// TIA Portal V19 export
FUNCTION_BLOCK "PositioningMachine_FB"   // FB24, LAD
TITLE = POSITIONING MACHINE
// stored: Access Published, MemoryReserve 100, SetENOAutomatically false
   VAR_INPUT
      AreaInterface : "AreaInterface";
      ZSI : "udt_ZoneSafetyInterface";
      DSI : "udt_DeviceSafetyInterface";
      Drive : "TAx_DriveInterface";
      DataIn : "PositioningMachine_DataIn";
      CIn : "PositioningMachine_CIn";
      Config : "PositioningMachine_Config";
      OL_CL_Space : LReal := 0.0;   // Limite rispetto allo spazio mancante per cambio da Move vel a Move pos abs
   END_VAR
   VAR_OUTPUT
      MachineInterface : "MachineInterface";
      DataOut : "PositioningMachine_DataOut";
      COut : "PositioningMachine_COut";
   END_VAR
   VAR_IN_OUT
      TO_Ax : TO_PositioningAxis;
      Par : "PositioningMachine_Par";
      Pers_Data : "PositioningMachine_DataPers";
      Warning : "PositioningMachine_Wng";
      Alarm : "PositioningMachine_Alr";
   END_VAR
   VAR
      InitDone : Bool := FALSE;
      Diag : Struct
         Ax : "TO_Diagnostic";
      END_STRUCT;
      HMI : Struct
         B_Preset : Bool;
         PresetPosition : LReal;
         TargetPosition : LReal;
      END_STRUCT;
      Sts : Struct
         Standstill : Bool := TRUE;
         AlarmPresence : Bool := FALSE;
         WarningPresence : Bool := FALSE;
         Man_UsePositionLimits : Bool;
         Aut_UsePositionLimits : Bool;
         Gen_Cnd : Bool;
         Bwd_Cnd : Bool := FALSE;
         Fwd_Cnd : Bool := FALSE;
         InTargetPosition : Bool;
         AxisModulo : LReal;
         MissingToTarget : LReal;
         MissingToTarget_ABS : LReal;
      END_STRUCT;
      Ctrl : Struct
         StopDueDoorOpeningRequest : Bool;
         StopInPhase : Bool;
         StopProgrammed : Bool;
         StopAborting : Bool;
         Man_HighSpeed : Bool;
         Bwd_Man : Bool;
         Fwd_Man : Bool;
         MoveToPos_Man : Bool;
         Bwd_Aut : Bool;
         Fwd_Aut : Bool;
         MoveToPos_Aut : Bool;
         Fan : Bool;
         Vel : LReal;
         Acc : LReal;
         Dec : LReal;
         Jerk : LReal;
      END_STRUCT;
      EncoderSelection { ExternalAccessible := 'False'; ExternalVisible := 'False'; ExternalWritable := 'False'} : "Axis_EncoderSelection_FB";
      WritePar { S7_SetPoint := 'True'} : "Axis_WritePar_FB";
      ReloadPosition { S7_SetPoint := 'True'} : "Axis_ReloadPosition_FB";
      LoadPosition : "Axis_ManPreset_FB";
      Ax { S7_SetPoint := 'True'} : "PositioningAxis";
      TorqueLimit { S7_SetPoint := 'True'} : MC_TORQUELIMITING;
      Fan_M : "Motor";
      TON_NoPendingCmd : TON_TIME;
      TON_Feed_DelayManChangeSpeed : TON_TIME;
      TON_InTargetPosition : TON_TIME;
      TON_MissingCndBwd { S7_SetPoint := 'True'} : TON_TIME;
      TON_MissingCndFwd { S7_SetPoint := 'True'} : TON_TIME;
      TON_Fan_DelayOff : TON_TIME;
      TON_Brake_TimeOut { S7_SetPoint := 'True'} : TON_TIME;
      AUX : Struct
         PB_Bwd : Bool;
         PB_Fwd : Bool;
         PB_MoveToPos : Bool;
         B_Preset : Bool;
      END_STRUCT;
   END_VAR
   VAR_TEMP
      PE : Struct
         PB_Bwd : Bool;
         PB_Fwd : Bool;
         PB_MoveToPos : Bool;
         B_Preset : Bool;
      END_STRUCT;
      Cnd : Bool;
      Req : Bool;
      Check : Bool;
      VelMaterialMover : LReal;
      RetVal_MeasWheelCheckRotation_Man : Int;
      RetVal_MeasWheelCheckRotation_Aut : Int;
      RetVal_MeasWheelCheckMechGearRatio : Int;
      MeasWheelVelOK : Bool;
      TorqueLimit_EngUnit : LReal;
      TorqueLimit_Percentage : LReal;
      TorqueLimit_DriveUnit : LReal;
      Bwd_CheckVel : Bool;
      Fwd_CheckVel : Bool;
      Bwd_CheckPos : Bool;
      Fwd_CheckPos : Bool;
      Real_VelTarget : LReal;
      RemainingDistanceABS : LReal;
      LimitExceeds : Bool;
      NegativeTolerance : LReal;
   END_VAR
   VAR_TEMP   // added for the SCL form of the ladder/FBD networks
      _w1 : Bool;
      _w2 : Bool;
      _w3 : Bool;
   END_VAR
BEGIN

REGION Network 1 (SCL): Init
   IF NOT #InitDone THEN

       #InitDone := TRUE;

       #Pers_Data.AxisEncoderSelection_OK := FALSE;

       #Pers_Data.AxisParameters_OK := FALSE;

       #Pers_Data.AxisReloadPostion_OK := FALSE;

   END_IF;
END_REGION

REGION Network 2 (SCL): Reset
   IF #AreaInterface.RstAlarms THEN

       #Alarm.AxisNotInOperation :=

       #Alarm.BrakeTimeOut :=

       #Warning.NotAutReady :=
       #Warning.AxisNotInOperation :=
       #Warning.MissingCnd_BWD :=
       #Warning.MissingCnd_FWD := FALSE;


   END_IF;
END_REGION

REGION Network 3: Alarm motor brake timeout
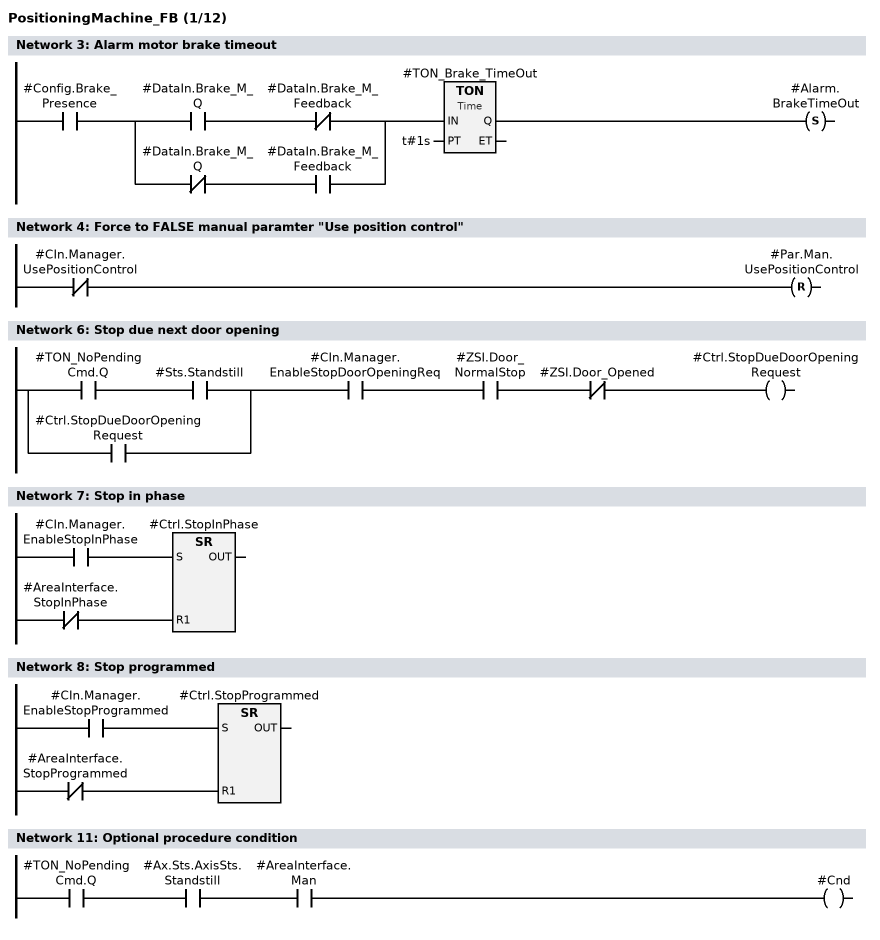
   RUNG wire#powerrail
      Contact( #Config.Brake_Presence )
      wire#w1
      Contact( #DataIn.Brake_M_Q )
      I_Contact( #DataIn.Brake_M_Feedback )
      wire#w2
      { S7_Templates := "time_type := Time" } #TON_Brake_TimeOut.TON(pt := t#1s, et =>)
      S_Coil( #Alarm.BrakeTimeOut )
   END_RUNG
   RUNG wire#w1
      I_Contact( #DataIn.Brake_M_Q )
      Contact( #DataIn.Brake_M_Feedback )
   END_RUNG wire#w2
   // the same network as SCL:
   #TON_Brake_TimeOut(IN := #Config.Brake_Presence AND ((#DataIn.Brake_M_Q AND NOT #DataIn.Brake_M_Feedback) OR (NOT #DataIn.Brake_M_Q AND #DataIn.Brake_M_Feedback)),   // TON
                      PT := t#1s);
   IF #TON_Brake_TimeOut.Q THEN #Alarm.BrakeTimeOut := TRUE; END_IF;
END_REGION

REGION Network 4: Force to FALSE manual paramter "Use position control"
   RUNG wire#powerrail
      I_Contact( #CIn.Manager.UsePositionControl )
      R_Coil( #Par.Man.UsePositionControl )
   END_RUNG
   // the same network as SCL:
   IF NOT #CIn.Manager.UsePositionControl THEN #Par.Man.UsePositionControl := FALSE; END_IF;
END_REGION

REGION Network 5: <<< MACHINE STOP >>>
END_REGION

REGION Network 6: Stop due next door opening
   RUNG wire#powerrail
      Contact( #TON_NoPendingCmd.Q )
      Contact( #Sts.Standstill )
      wire#w1
      Contact( #CIn.Manager.EnableStopDoorOpeningReq )
      Contact( #ZSI.Door_NormalStop )
      I_Contact( #ZSI.Door_Opened )
      Coil( #Ctrl.StopDueDoorOpeningRequest )
   END_RUNG
   RUNG wire#powerrail
      Contact( #Ctrl.StopDueDoorOpeningRequest )
   END_RUNG wire#w1
   // the same network as SCL:
   #Ctrl.StopDueDoorOpeningRequest := ((#TON_NoPendingCmd.Q AND #Sts.Standstill) OR #Ctrl.StopDueDoorOpeningRequest) AND #CIn.Manager.EnableStopDoorOpeningReq AND #ZSI.Door_NormalStop AND NOT #ZSI.Door_Opened;
END_REGION

REGION Network 7: Stop in phase
   RUNG wire#powerrail
      Contact( #CIn.Manager.EnableStopInPhase )
      S_SR(operand := #Ctrl.StopInPhase, r1 := wire#w1)
   END_RUNG
   RUNG wire#powerrail
      I_Contact( #AreaInterface.StopInPhase )
   END_RUNG wire#w1
   // the same network as SCL:
   IF #CIn.Manager.EnableStopInPhase THEN
       #Ctrl.StopInPhase := TRUE;   // SR flip-flop
   END_IF;
   IF NOT #AreaInterface.StopInPhase THEN #Ctrl.StopInPhase := FALSE; END_IF;
END_REGION

REGION Network 8: Stop programmed
   RUNG wire#powerrail
      Contact( #CIn.Manager.EnableStopProgrammed )
      S_SR(operand := #Ctrl.StopProgrammed, r1 := wire#w1)
   END_RUNG
   RUNG wire#powerrail
      I_Contact( #AreaInterface.StopProgrammed )
   END_RUNG wire#w1
   // the same network as SCL:
   IF #CIn.Manager.EnableStopProgrammed THEN
       #Ctrl.StopProgrammed := TRUE;   // SR flip-flop
   END_IF;
   IF NOT #AreaInterface.StopProgrammed THEN #Ctrl.StopProgrammed := FALSE; END_IF;
END_REGION

REGION Network 9: >
END_REGION

REGION Network 10: <<< OPTIONS >>>
END_REGION

REGION Network 11: Optional procedure condition
   RUNG wire#powerrail
      Contact( #TON_NoPendingCmd.Q )
      Contact( #Ax.Sts.AxisSts.Standstill )
      Contact( #AreaInterface.Man )
      Coil( #Cnd )
   END_RUNG
   // the same network as SCL:
   #Cnd := #TON_NoPendingCmd.Q AND #Ax.Sts.AxisSts.Standstill AND #AreaInterface.Man;
END_REGION

REGION Network 12: (OPTION) Motor / Measuring wheel encoder exchange
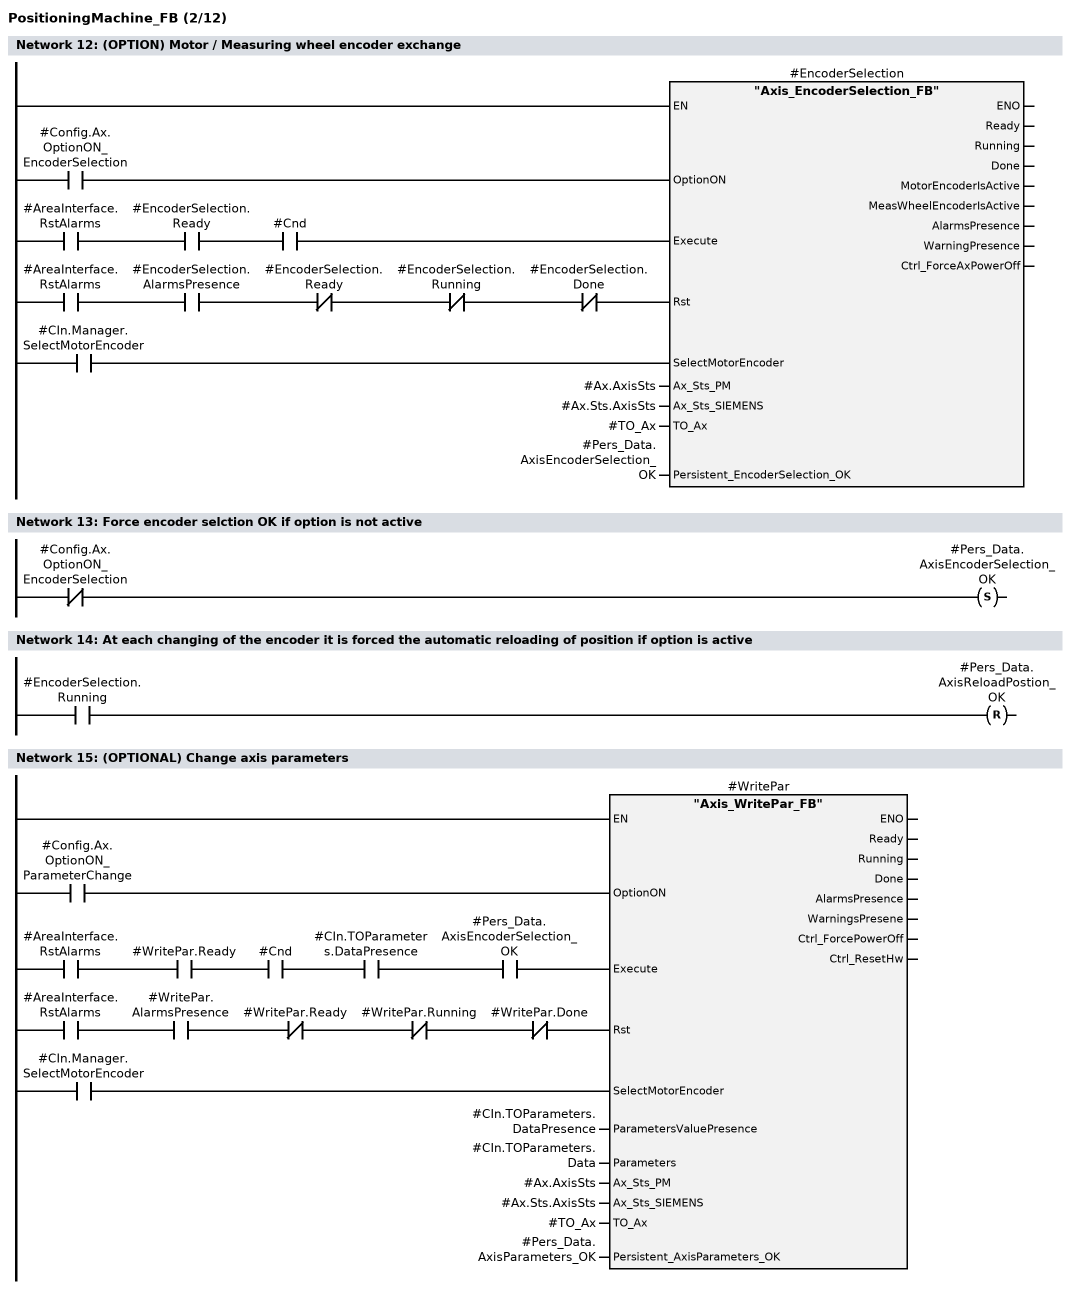
   RUNG wire#powerrail
      #EncoderSelection(OptionON := wire#w1, Execute := wire#w2, Rst := wire#w3, SelectMotorEncoder := wire#w4, Ax_Sts_PM := #Ax.AxisSts, Ax_Sts_SIEMENS := #Ax.Sts.AxisSts, TO_Ax := #TO_Ax, Persistent_EncoderSelection_OK := #Pers_Data.AxisEncoderSelection_OK, Ready =>, Running =>, Done =>, MotorEncoderIsActive =>, MeasWheelEncoderIsActive =>, AlarmsPresence =>, WarningPresence =>, Ctrl_ForceAxPowerOff =>)
   END_RUNG
   RUNG wire#powerrail
      Contact( #Config.Ax.OptionON_EncoderSelection )
   END_RUNG wire#w1
   RUNG wire#powerrail
      Contact( #AreaInterface.RstAlarms )
      Contact( #EncoderSelection.Ready )
      Contact( #Cnd )
   END_RUNG wire#w2
   RUNG wire#powerrail
      Contact( #AreaInterface.RstAlarms )
      Contact( #EncoderSelection.AlarmsPresence )
      I_Contact( #EncoderSelection.Ready )
      I_Contact( #EncoderSelection.Running )
      I_Contact( #EncoderSelection.Done )
   END_RUNG wire#w3
   RUNG wire#powerrail
      Contact( #CIn.Manager.SelectMotorEncoder )
   END_RUNG wire#w4
   // the same network as SCL:
   #EncoderSelection(OptionON := #Config.Ax.OptionON_EncoderSelection,   // "Axis_EncoderSelection_FB"
                     Execute := #AreaInterface.RstAlarms AND #EncoderSelection.Ready AND #Cnd,
                     Rst := #AreaInterface.RstAlarms AND #EncoderSelection.AlarmsPresence AND NOT #EncoderSelection.Ready AND NOT #EncoderSelection.Running AND NOT #EncoderSelection.Done,
                     SelectMotorEncoder := #CIn.Manager.SelectMotorEncoder,
                     Ax_Sts_PM := #Ax.AxisSts,
                     Ax_Sts_SIEMENS := #Ax.Sts.AxisSts,
                     TO_Ax := #TO_Ax,
                     Persistent_EncoderSelection_OK := #Pers_Data.AxisEncoderSelection_OK);
END_REGION

REGION Network 13: Force encoder selction OK if option is not active
   RUNG wire#powerrail
      I_Contact( #Config.Ax.OptionON_EncoderSelection )
      S_Coil( #Pers_Data.AxisEncoderSelection_OK )
   END_RUNG
   // the same network as SCL:
   IF NOT #Config.Ax.OptionON_EncoderSelection THEN #Pers_Data.AxisEncoderSelection_OK := TRUE; END_IF;
END_REGION

REGION Network 14: At each changing of the encoder it is forced the automatic reloading of position if option is active
   RUNG wire#powerrail
      Contact( #EncoderSelection.Running )
      R_Coil( #Pers_Data.AxisReloadPostion_OK )
   END_RUNG
   // the same network as SCL:
   IF #EncoderSelection.Running THEN #Pers_Data.AxisReloadPostion_OK := FALSE; END_IF;
END_REGION

REGION Network 15: (OPTIONAL) Change axis parameters
   RUNG wire#powerrail
      #WritePar(OptionON := wire#w1, Execute := wire#w2, Rst := wire#w3, SelectMotorEncoder := wire#w4, ParametersValuePresence := #CIn.TOParameters.DataPresence, Parameters := #CIn.TOParameters.Data, Ax_Sts_PM := #Ax.AxisSts, Ax_Sts_SIEMENS := #Ax.Sts.AxisSts, TO_Ax := #TO_Ax, Persistent_AxisParameters_OK := #Pers_Data.AxisParameters_OK, Ready =>, Running =>, Done =>, AlarmsPresence =>, WarningsPresene =>, Ctrl_ForcePowerOff =>, Ctrl_ResetHw =>)
   END_RUNG
   RUNG wire#powerrail
      Contact( #Config.Ax.OptionON_ParameterChange )
   END_RUNG wire#w1
   RUNG wire#powerrail
      Contact( #AreaInterface.RstAlarms )
      Contact( #WritePar.Ready )
      Contact( #Cnd )
      Contact( #CIn.TOParameters.DataPresence )
      Contact( #Pers_Data.AxisEncoderSelection_OK )
   END_RUNG wire#w2
   RUNG wire#powerrail
      Contact( #AreaInterface.RstAlarms )
      Contact( #WritePar.AlarmsPresence )
      I_Contact( #WritePar.Ready )
      I_Contact( #WritePar.Running )
      I_Contact( #WritePar.Done )
   END_RUNG wire#w3
   RUNG wire#powerrail
      Contact( #CIn.Manager.SelectMotorEncoder )
   END_RUNG wire#w4
   // the same network as SCL:
   #WritePar(OptionON := #Config.Ax.OptionON_ParameterChange,   // "Axis_WritePar_FB"
             Execute := #AreaInterface.RstAlarms AND #WritePar.Ready AND #Cnd AND #CIn.TOParameters.DataPresence AND #Pers_Data.AxisEncoderSelection_OK,
             Rst := #AreaInterface.RstAlarms AND #WritePar.AlarmsPresence AND NOT #WritePar.Ready AND NOT #WritePar.Running AND NOT #WritePar.Done,
             SelectMotorEncoder := #CIn.Manager.SelectMotorEncoder,
             ParametersValuePresence := #CIn.TOParameters.DataPresence,
             Parameters := #CIn.TOParameters.Data,
             Ax_Sts_PM := #Ax.AxisSts,
             Ax_Sts_SIEMENS := #Ax.Sts.AxisSts,
             TO_Ax := #TO_Ax,
             Persistent_AxisParameters_OK := #Pers_Data.AxisParameters_OK);
END_REGION

REGION Network 16: Force parameter write execution ok if option is not active
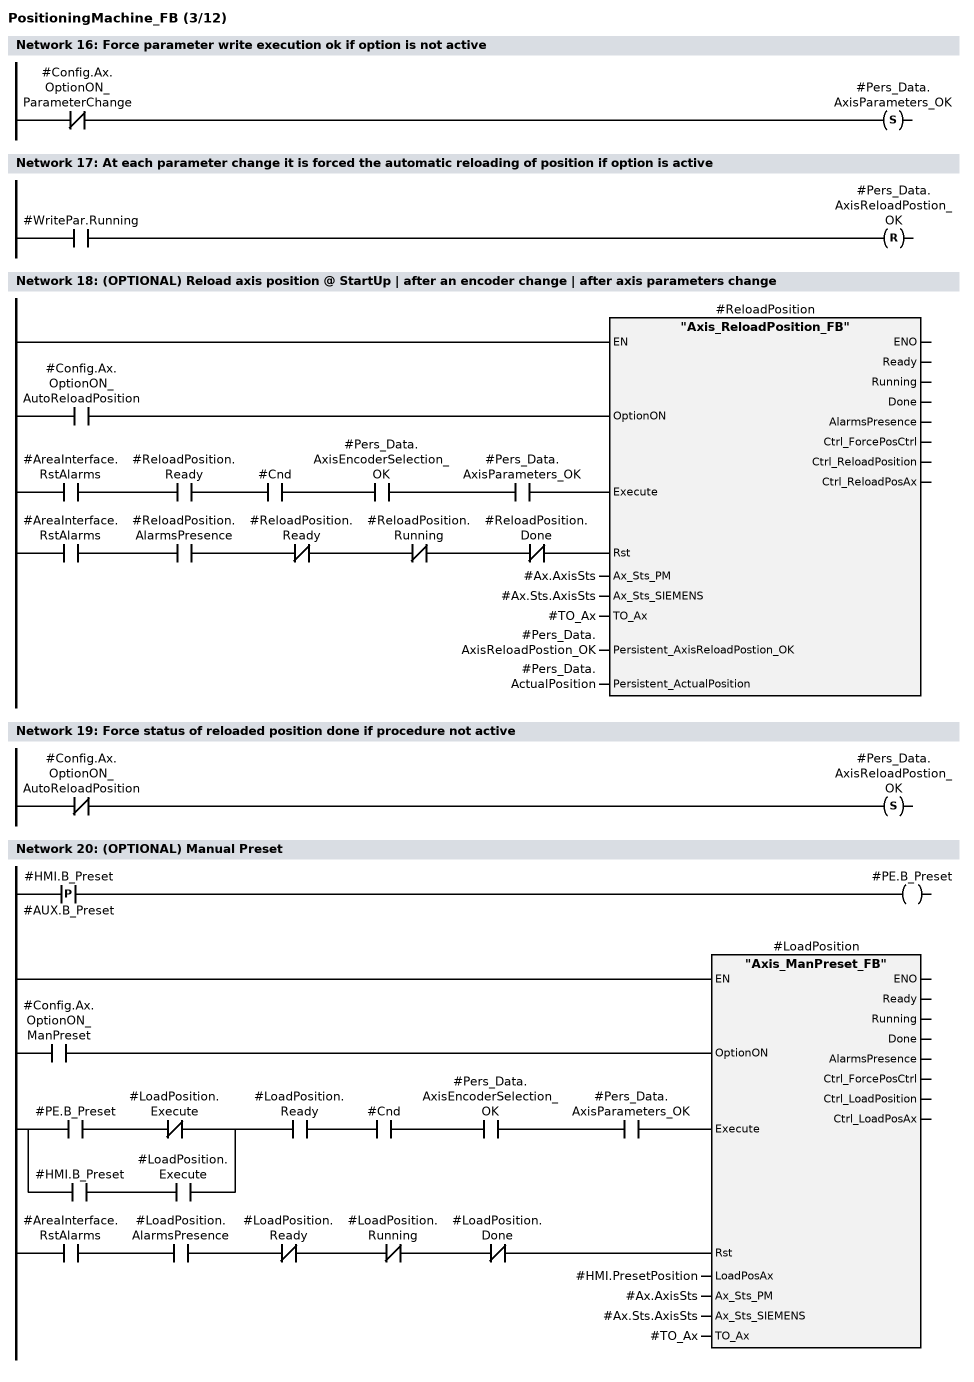
   RUNG wire#powerrail
      I_Contact( #Config.Ax.OptionON_ParameterChange )
      S_Coil( #Pers_Data.AxisParameters_OK )
   END_RUNG
   // the same network as SCL:
   IF NOT #Config.Ax.OptionON_ParameterChange THEN #Pers_Data.AxisParameters_OK := TRUE; END_IF;
END_REGION

REGION Network 17: At each parameter change it is forced the automatic reloading of position if option is active
   RUNG wire#powerrail
      Contact( #WritePar.Running )
      R_Coil( #Pers_Data.AxisReloadPostion_OK )
   END_RUNG
   // the same network as SCL:
   IF #WritePar.Running THEN #Pers_Data.AxisReloadPostion_OK := FALSE; END_IF;
END_REGION

REGION Network 18: (OPTIONAL) Reload axis position @ StartUp | after an encoder change | after axis parameters change
   RUNG wire#powerrail
      #ReloadPosition(OptionON := wire#w1, Execute := wire#w2, Rst := wire#w3, Ax_Sts_PM := #Ax.AxisSts, Ax_Sts_SIEMENS := #Ax.Sts.AxisSts, TO_Ax := #TO_Ax, Persistent_AxisReloadPostion_OK := #Pers_Data.AxisReloadPostion_OK, Persistent_ActualPosition := #Pers_Data.ActualPosition, Ready =>, Running =>, Done =>, AlarmsPresence =>, Ctrl_ForcePosCtrl =>, Ctrl_ReloadPosition =>, Ctrl_ReloadPosAx =>)
   END_RUNG
   RUNG wire#powerrail
      Contact( #Config.Ax.OptionON_AutoReloadPosition )
   END_RUNG wire#w1
   RUNG wire#powerrail
      Contact( #AreaInterface.RstAlarms )
      Contact( #ReloadPosition.Ready )
      Contact( #Cnd )
      Contact( #Pers_Data.AxisEncoderSelection_OK )
      Contact( #Pers_Data.AxisParameters_OK )
   END_RUNG wire#w2
   RUNG wire#powerrail
      Contact( #AreaInterface.RstAlarms )
      Contact( #ReloadPosition.AlarmsPresence )
      I_Contact( #ReloadPosition.Ready )
      I_Contact( #ReloadPosition.Running )
      I_Contact( #ReloadPosition.Done )
   END_RUNG wire#w3
   // the same network as SCL:
   #ReloadPosition(OptionON := #Config.Ax.OptionON_AutoReloadPosition,   // "Axis_ReloadPosition_FB"
                   Execute := #AreaInterface.RstAlarms AND #ReloadPosition.Ready AND #Cnd AND #Pers_Data.AxisEncoderSelection_OK AND #Pers_Data.AxisParameters_OK,
                   Rst := #AreaInterface.RstAlarms AND #ReloadPosition.AlarmsPresence AND NOT #ReloadPosition.Ready AND NOT #ReloadPosition.Running AND NOT #ReloadPosition.Done,
                   Ax_Sts_PM := #Ax.AxisSts,
                   Ax_Sts_SIEMENS := #Ax.Sts.AxisSts,
                   TO_Ax := #TO_Ax,
                   Persistent_AxisReloadPostion_OK := #Pers_Data.AxisReloadPostion_OK,
                   Persistent_ActualPosition := #Pers_Data.ActualPosition);
END_REGION

REGION Network 19: Force status of reloaded position done if procedure not active
   RUNG wire#powerrail
      I_Contact( #Config.Ax.OptionON_AutoReloadPosition )
      S_Coil( #Pers_Data.AxisReloadPostion_OK )
   END_RUNG
   // the same network as SCL:
   IF NOT #Config.Ax.OptionON_AutoReloadPosition THEN #Pers_Data.AxisReloadPostion_OK := TRUE; END_IF;
END_REGION

REGION Network 20: (OPTIONAL) Manual Preset
   RUNG wire#powerrail
      P_Contact(operand := #HMI.B_Preset, bit := #AUX.B_Preset)
      Coil( #PE.B_Preset )
   END_RUNG
   RUNG wire#powerrail
      #LoadPosition(OptionON := wire#w1, Execute := wire#w3, Rst := wire#w4, LoadPosAx := #HMI.PresetPosition, Ax_Sts_PM := #Ax.AxisSts, Ax_Sts_SIEMENS := #Ax.Sts.AxisSts, TO_Ax := #TO_Ax, Ready =>, Running =>, Done =>, AlarmsPresence =>, Ctrl_ForcePosCtrl =>, Ctrl_LoadPosition =>, Ctrl_LoadPosAx =>)
   END_RUNG
   RUNG wire#powerrail
      Contact( #Config.Ax.OptionON_ManPreset )
   END_RUNG wire#w1
   RUNG wire#powerrail
      Contact( #PE.B_Preset )
      I_Contact( #LoadPosition.Execute )
      wire#w2
      Contact( #LoadPosition.Ready )
      Contact( #Cnd )
      Contact( #Pers_Data.AxisEncoderSelection_OK )
      Contact( #Pers_Data.AxisParameters_OK )
   END_RUNG wire#w3
   RUNG wire#powerrail
      Contact( #HMI.B_Preset )
      Contact( #LoadPosition.Execute )
   END_RUNG wire#w2
   RUNG wire#powerrail
      Contact( #AreaInterface.RstAlarms )
      Contact( #LoadPosition.AlarmsPresence )
      I_Contact( #LoadPosition.Ready )
      I_Contact( #LoadPosition.Running )
      I_Contact( #LoadPosition.Done )
   END_RUNG wire#w4
   // the same network as SCL:
   #_w1 := #HMI.B_Preset AND NOT #AUX.B_Preset;   // rising edge of #HMI.B_Preset
   #AUX.B_Preset := #HMI.B_Preset;
   #PE.B_Preset := #_w1;
   #LoadPosition(OptionON := #Config.Ax.OptionON_ManPreset,   // "Axis_ManPreset_FB"
                 Execute := ((#PE.B_Preset AND NOT #LoadPosition.Execute) OR (#HMI.B_Preset AND #LoadPosition.Execute)) AND #LoadPosition.Ready AND #Cnd AND #Pers_Data.AxisEncoderSelection_OK AND #Pers_Data.AxisParameters_OK,
                 Rst := #AreaInterface.RstAlarms AND #LoadPosition.AlarmsPresence AND NOT #LoadPosition.Ready AND NOT #LoadPosition.Running AND NOT #LoadPosition.Done,
                 LoadPosAx := #HMI.PresetPosition,
                 Ax_Sts_PM := #Ax.AxisSts,
                 Ax_Sts_SIEMENS := #Ax.Sts.AxisSts,
                 TO_Ax := #TO_Ax);
END_REGION

REGION Network 21: At each Load position done Set Reloaad position OK
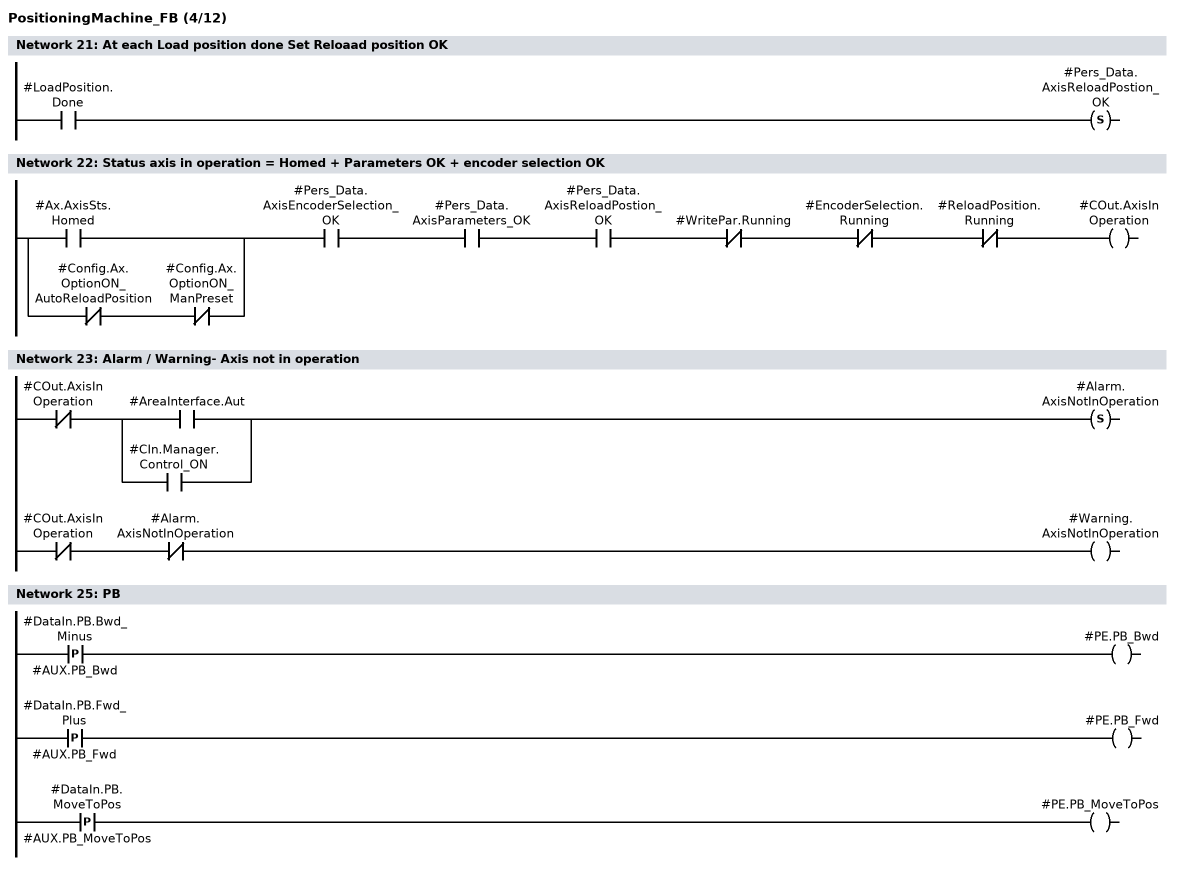
   RUNG wire#powerrail
      Contact( #LoadPosition.Done )
      S_Coil( #Pers_Data.AxisReloadPostion_OK )
   END_RUNG
   // the same network as SCL:
   IF #LoadPosition.Done THEN #Pers_Data.AxisReloadPostion_OK := TRUE; END_IF;
END_REGION

REGION Network 22: Status axis in operation = Homed + Parameters OK + encoder selection OK
   RUNG wire#powerrail
      Contact( #Ax.AxisSts.Homed )
      wire#w1
      Contact( #Pers_Data.AxisEncoderSelection_OK )
      Contact( #Pers_Data.AxisParameters_OK )
      Contact( #Pers_Data.AxisReloadPostion_OK )
      I_Contact( #WritePar.Running )
      I_Contact( #EncoderSelection.Running )
      I_Contact( #ReloadPosition.Running )
      Coil( #COut.AxisInOperation )
   END_RUNG
   RUNG wire#powerrail
      I_Contact( #Config.Ax.OptionON_AutoReloadPosition )
      I_Contact( #Config.Ax.OptionON_ManPreset )
   END_RUNG wire#w1
   // the same network as SCL:
   #COut.AxisInOperation := (#Ax.AxisSts.Homed OR (NOT #Config.Ax.OptionON_AutoReloadPosition AND NOT #Config.Ax.OptionON_ManPreset)) AND #Pers_Data.AxisEncoderSelection_OK AND #Pers_Data.AxisParameters_OK AND #Pers_Data.AxisReloadPostion_OK AND NOT #WritePar.Running AND NOT #EncoderSelection.Running AND NOT #ReloadPosition.Running;
END_REGION

REGION Network 23: Alarm / Warning- Axis not in operation
   RUNG wire#powerrail
      I_Contact( #COut.AxisInOperation )
      wire#w1
      Contact( #AreaInterface.Aut )
      wire#w2
      S_Coil( #Alarm.AxisNotInOperation )
   END_RUNG
   RUNG wire#w1
      Contact( #CIn.Manager.Control_ON )
   END_RUNG wire#w2
   RUNG wire#powerrail
      I_Contact( #COut.AxisInOperation )
      I_Contact( #Alarm.AxisNotInOperation )
      Coil( #Warning.AxisNotInOperation )
   END_RUNG
   // the same network as SCL:
   IF NOT #COut.AxisInOperation AND (#AreaInterface.Aut OR #CIn.Manager.Control_ON) THEN
       #Alarm.AxisNotInOperation := TRUE;
   END_IF;
   #Warning.AxisNotInOperation := NOT #COut.AxisInOperation AND NOT #Alarm.AxisNotInOperation;
END_REGION

REGION Network 24: <<< FEED >>>
END_REGION

REGION Network 25: PB
   RUNG wire#powerrail
      P_Contact(operand := #DataIn.PB.Bwd_Minus, bit := #AUX.PB_Bwd)
      Coil( #PE.PB_Bwd )
   END_RUNG
   RUNG wire#powerrail
      P_Contact(operand := #DataIn.PB.Fwd_Plus, bit := #AUX.PB_Fwd)
      Coil( #PE.PB_Fwd )
   END_RUNG
   RUNG wire#powerrail
      P_Contact(operand := #DataIn.PB.MoveToPos, bit := #AUX.PB_MoveToPos)
      Coil( #PE.PB_MoveToPos )
   END_RUNG
   // the same network as SCL:
   #_w1 := #DataIn.PB.Bwd_Minus AND NOT #AUX.PB_Bwd;   // rising edge of #DataIn.PB.Bwd_Minus
   #AUX.PB_Bwd := #DataIn.PB.Bwd_Minus;
   #PE.PB_Bwd := #_w1;
   #_w2 := #DataIn.PB.Fwd_Plus AND NOT #AUX.PB_Fwd;   // rising edge of #DataIn.PB.Fwd_Plus
   #AUX.PB_Fwd := #DataIn.PB.Fwd_Plus;
   #PE.PB_Fwd := #_w2;
   #_w3 := #DataIn.PB.MoveToPos AND NOT #AUX.PB_MoveToPos;   // rising edge of #DataIn.PB.MoveToPos
   #AUX.PB_MoveToPos := #DataIn.PB.MoveToPos;
   #PE.PB_MoveToPos := #_w3;
END_REGION

REGION Network 26: Man
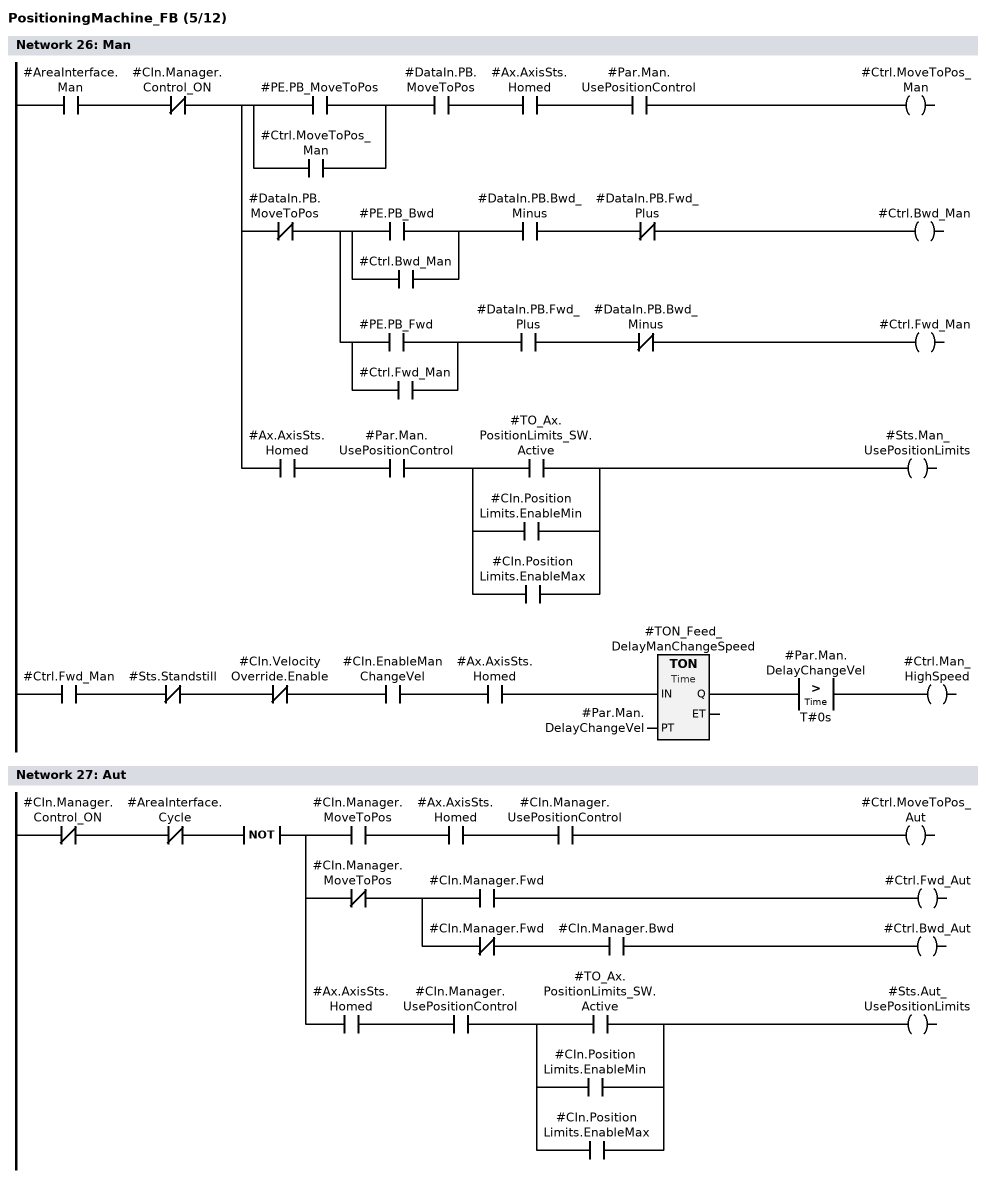
   RUNG wire#powerrail
      Contact( #AreaInterface.Man )
      I_Contact( #CIn.Manager.Control_ON )
      wire#w1
      Contact( #PE.PB_MoveToPos )
      wire#w2
      Contact( #DataIn.PB.MoveToPos )
      Contact( #Ax.AxisSts.Homed )
      Contact( #Par.Man.UsePositionControl )
      Coil( #Ctrl.MoveToPos_Man )
   END_RUNG
   RUNG wire#w1
      Contact( #Ctrl.MoveToPos_Man )
   END_RUNG wire#w2
   RUNG wire#w1
      I_Contact( #DataIn.PB.MoveToPos )
      wire#w3
      Contact( #PE.PB_Bwd )
      wire#w4
      Contact( #DataIn.PB.Bwd_Minus )
      I_Contact( #DataIn.PB.Fwd_Plus )
      Coil( #Ctrl.Bwd_Man )
   END_RUNG
   RUNG wire#w3
      Contact( #Ctrl.Bwd_Man )
   END_RUNG wire#w4
   RUNG wire#w3
      Contact( #PE.PB_Fwd )
      wire#w5
      Contact( #DataIn.PB.Fwd_Plus )
      I_Contact( #DataIn.PB.Bwd_Minus )
      Coil( #Ctrl.Fwd_Man )
   END_RUNG
   RUNG wire#w3
      Contact( #Ctrl.Fwd_Man )
   END_RUNG wire#w5
   RUNG wire#w1
      Contact( #Ax.AxisSts.Homed )
      Contact( #Par.Man.UsePositionControl )
      wire#w6
      Contact( #TO_Ax.PositionLimits_SW.Active )
      wire#w7
      Coil( #Sts.Man_UsePositionLimits )
   END_RUNG
   RUNG wire#w6
      Contact( #CIn.PositionLimits.EnableMin )
   END_RUNG wire#w7
   RUNG wire#w6
      Contact( #CIn.PositionLimits.EnableMax )
   END_RUNG wire#w7
   RUNG wire#powerrail
      Contact( #Ctrl.Fwd_Man )
      I_Contact( #Sts.Standstill )
      I_Contact( #CIn.VelocityOverride.Enable )
      Contact( #CIn.EnableManChangeVel )
      Contact( #Ax.AxisSts.Homed )
      { S7_Templates := "time_type := Time" } #TON_Feed_DelayManChangeSpeed.TON(pt := #Par.Man.DelayChangeVel, et =>)
      { S7_Templates := "SrcType := Time" } GT_Contact(in1 := #Par.Man.DelayChangeVel, in2 := T#0s)
      Coil( #Ctrl.Man_HighSpeed )
   END_RUNG
   // the same network as SCL:
   #_w1 := #AreaInterface.Man AND NOT #CIn.Manager.Control_ON;
   #Ctrl.MoveToPos_Man := #_w1 AND (#PE.PB_MoveToPos OR #Ctrl.MoveToPos_Man) AND #DataIn.PB.MoveToPos AND #Ax.AxisSts.Homed AND #Par.Man.UsePositionControl;
   #_w2 := #_w1 AND NOT #DataIn.PB.MoveToPos;
   #Ctrl.Bwd_Man := #_w2 AND (#PE.PB_Bwd OR #Ctrl.Bwd_Man) AND #DataIn.PB.Bwd_Minus AND NOT #DataIn.PB.Fwd_Plus;
   #Ctrl.Fwd_Man := #_w2 AND (#PE.PB_Fwd OR #Ctrl.Fwd_Man) AND #DataIn.PB.Fwd_Plus AND NOT #DataIn.PB.Bwd_Minus;
   #Sts.Man_UsePositionLimits := #_w1 AND #Ax.AxisSts.Homed AND #Par.Man.UsePositionControl AND (#TO_Ax.PositionLimits_SW.Active OR #CIn.PositionLimits.EnableMin OR #CIn.PositionLimits.EnableMax);
   #TON_Feed_DelayManChangeSpeed(IN := #Ctrl.Fwd_Man AND NOT #Sts.Standstill AND NOT #CIn.VelocityOverride.Enable AND #CIn.EnableManChangeVel AND #Ax.AxisSts.Homed,   // TON
                           PT := #Par.Man.DelayChangeVel);
   #Ctrl.Man_HighSpeed := #TON_Feed_DelayManChangeSpeed.Q AND (#Par.Man.DelayChangeVel > T#0s);
END_REGION

REGION Network 27: Aut
   RUNG wire#powerrail
      I_Contact( #CIn.Manager.Control_ON )
      I_Contact( #AreaInterface.Cycle )
      Not()
      wire#w1
      Contact( #CIn.Manager.MoveToPos )
      Contact( #Ax.AxisSts.Homed )
      Contact( #CIn.Manager.UsePositionControl )
      Coil( #Ctrl.MoveToPos_Aut )
   END_RUNG
   RUNG wire#w1
      I_Contact( #CIn.Manager.MoveToPos )
      wire#w2
      Contact( #CIn.Manager.Fwd )
      Coil( #Ctrl.Fwd_Aut )
   END_RUNG
   RUNG wire#w2
      I_Contact( #CIn.Manager.Fwd )
      Contact( #CIn.Manager.Bwd )
      Coil( #Ctrl.Bwd_Aut )
   END_RUNG
   RUNG wire#w1
      Contact( #Ax.AxisSts.Homed )
      Contact( #CIn.Manager.UsePositionControl )
      wire#w3
      Contact( #TO_Ax.PositionLimits_SW.Active )
      wire#w4
      Coil( #Sts.Aut_UsePositionLimits )
   END_RUNG
   RUNG wire#w3
      Contact( #CIn.PositionLimits.EnableMin )
   END_RUNG wire#w4
   RUNG wire#w3
      Contact( #CIn.PositionLimits.EnableMax )
   END_RUNG wire#w4
   // the same network as SCL:
   #_w1 := NOT (NOT #CIn.Manager.Control_ON AND NOT #AreaInterface.Cycle);
   #Ctrl.MoveToPos_Aut := #_w1 AND #CIn.Manager.MoveToPos AND #Ax.AxisSts.Homed AND #CIn.Manager.UsePositionControl;
   #_w2 := #_w1 AND NOT #CIn.Manager.MoveToPos;
   #Ctrl.Fwd_Aut := #_w2 AND #CIn.Manager.Fwd;
   #Ctrl.Bwd_Aut := #_w2 AND NOT #CIn.Manager.Fwd AND #CIn.Manager.Bwd;
   #Sts.Aut_UsePositionLimits := #_w1 AND #Ax.AxisSts.Homed AND #CIn.Manager.UsePositionControl AND (#TO_Ax.PositionLimits_SW.Active OR #CIn.PositionLimits.EnableMin OR #CIn.PositionLimits.EnableMax);
END_REGION

REGION Network 28: >
END_REGION

REGION Network 29 (SCL): Axis Modulo value; 0 If isn't a modulo axis
   #Sts.AxisModulo := 0.0;

   IF #TO_Ax.Modulo.Enable THEN
       #Sts.AxisModulo := #TO_Ax.Modulo.Length - #TO_Ax.Modulo.StartValue;
   END_IF;
END_REGION

REGION Network 30 (SCL): Position Limits
   IF #Sts.AxisModulo > 0.0 THEN

       #COut.MinPosition := #Sts.AxisModulo * 5;
       #COut.MaxPosition := #Sts.AxisModulo * 5;
   ELSE

       #COut.MinPosition := -999999999.99;
       #COut.MaxPosition := +999999999.99;

   END_IF;



   #COut.BwdMinusLsSwReached := FALSE;
   #COut.FwdPlusLsSwReached := FALSE;

   #COut.BwdMinusLimitReached := FALSE;
   #COut.FwdPlusLimitReached := FALSE;



   IF #Ax.AxisSts.Homed THEN


       //.. If software limits are enabled...
       //
       IF #TO_Ax.PositionLimits_SW.Active THEN


           // Software limit Minus reached or exceeds
           // 
           #RemainingDistanceABS := ABS("M_PosAMinusPosB"(PosA := #Pers_Data.ActualPosition, PosB := #TO_Ax.PositionLimits_SW.MinPosition, MODULE := #Sts.AxisModulo));

           #LimitExceeds := "M_CmpLT"(Xa := #Pers_Data.ActualPosition, Xb := #TO_Ax.PositionLimits_SW.MinPosition, MODULE := #Sts.AxisModulo);

           #COut.BwdMinusLsSwReached := (#RemainingDistanceABS <= #Par.PosTolerance) OR #LimitExceeds;


           // Software limit Plus reached or exceeds
           // 
           #RemainingDistanceABS := ABS("M_PosAMinusPosB"(PosA := #Pers_Data.ActualPosition, PosB := #TO_Ax.PositionLimits_SW.MaxPosition, MODULE := #Sts.AxisModulo));

           #LimitExceeds := "M_CmpGT"(Xa := #Pers_Data.ActualPosition, Xb := #TO_Ax.PositionLimits_SW.MaxPosition, MODULE := #Sts.AxisModulo);

           #COut.FwdPlusLsSwReached := (#RemainingDistanceABS <= #Par.PosTolerance) OR #LimitExceeds;



           // Set general Min / Max position limit
           // 
           #COut.MinPosition := "M_PosAPlusCostB"(PosA := #TO_Ax.PositionLimits_SW.MinPosition, CostB := (#Par.PosTolerance / 2), MODULE := #Sts.AxisModulo);
           #COut.MaxPosition := "M_PosAMinusCostB"(PosA := #TO_Ax.PositionLimits_SW.MaxPosition, CostB := (#Par.PosTolerance / 2), MODULE := #Sts.AxisModulo);

       END_IF;

       //.. IF dynamic MIN limit set..
       //
       IF #CIn.PositionLimits.EnableMin
       THEN


           #RemainingDistanceABS := ABS("M_PosAMinusPosB"(PosA := #Pers_Data.ActualPosition, PosB := #CIn.PositionLimits.PosMin, MODULE := #Sts.AxisModulo));

           #LimitExceeds := "M_CmpLT"(Xa := #Pers_Data.ActualPosition, Xb := #CIn.PositionLimits.PosMin, MODULE := #Sts.AxisModulo);

           #COut.BwdMinusLimitReached := (#RemainingDistanceABS <= #Par.PosTolerance) OR #LimitExceeds;

           // Update general MIN limit
           // 
           IF "M_CmpGT"(Xa := #CIn.PositionLimits.PosMin, Xb := #COut.MinPosition, MODULE := #Sts.AxisModulo)
           THEN
               #COut.MinPosition := #CIn.PositionLimits.PosMin;
           END_IF;
       END_IF;


       //.. IF dynamic MAX limit set..
       //
       IF #CIn.PositionLimits.EnableMax
       THEN

           #RemainingDistanceABS := ABS("M_PosAMinusPosB"(PosA := #Pers_Data.ActualPosition, PosB := #CIn.PositionLimits.PosMax, MODULE := #Sts.AxisModulo));

           #LimitExceeds := "M_CmpGT"(Xa := #Pers_Data.ActualPosition, Xb := #CIn.PositionLimits.PosMax, MODULE := #Sts.AxisModulo);

           #COut.FwdPlusLimitReached := (#RemainingDistanceABS <= #Par.PosTolerance) OR #LimitExceeds;


           // Update general MAX limit
           // 
           IF "M_CmpLT"(Xa := #CIn.PositionLimits.PosMax, Xb := #COut.MaxPosition, MODULE := #Sts.AxisModulo)
           THEN
               #COut.MaxPosition := #CIn.PositionLimits.PosMax;
           END_IF;

       END_IF;




       IF #CIn.PositionLimits.EnableMin THEN
           #COut.MinPosition := MAX(IN1 := #COut.MinPosition, IN2 := #CIn.PositionLimits.PosMin);
       END_IF;


       IF #CIn.PositionLimits.EnableMax THEN
           #COut.MaxPosition := MIN(IN1 := #COut.MaxPosition, IN2 := #CIn.PositionLimits.PosMax);
       END_IF;

   END_IF;
END_REGION

REGION Network 31 (SCL): Axis Control (Target position)
   // Move Abs parameters
   // 
   #Ax.AxisCtrl.MoveAbsDirection := 3;


   // Target position choose
   // 

   IF #CIn.Manager.Control_ON THEN

       #Ax.AxisCtrl.MoveAbsTarget := #CIn.Manager.Pos;


       IF #Ctrl.Bwd_Aut AND #Sts.Aut_UsePositionLimits THEN

           #Ax.AxisCtrl.MoveAbsTarget := #COut.MinPosition;

       ELSIF #Ctrl.Fwd_Aut AND #Sts.Aut_UsePositionLimits THEN

           #Ax.AxisCtrl.MoveAbsTarget := #COut.MinPosition;
       END_IF;

       #HMI.TargetPosition := #Ax.AxisCtrl.MoveAbsTarget;


   ELSIF #Ctrl.MoveToPos_Man  THEN

       #Ax.AxisCtrl.MoveAbsTarget := #HMI.TargetPosition;


   ELSIF #Ctrl.Bwd_Man AND #Sts.Man_UsePositionLimits THEN

       #Ax.AxisCtrl.MoveAbsTarget := #COut.MinPosition;
       #HMI.TargetPosition := #Ax.AxisCtrl.MoveAbsTarget;

   ELSIF #Ctrl.Fwd_Man AND #Sts.Man_UsePositionLimits THEN

       #Ax.AxisCtrl.MoveAbsTarget := #COut.MaxPosition;
       #HMI.TargetPosition := #Ax.AxisCtrl.MoveAbsTarget;

   END_IF;


   // Check Target position within limits
   //

   IF #Sts.Man_UsePositionLimits OR #Sts.Aut_UsePositionLimits THEN


       // Target position exceeds MIN limit
       // 
       #LimitExceeds := "M_CmpLT"(Xa := #Ax.AxisCtrl.MoveAbsTarget, Xb := #COut.MinPosition, MODULE := #Sts.AxisModulo);
       IF #LimitExceeds THEN
           #Ax.AxisCtrl.MoveAbsTarget := #COut.MinPosition;
           #HMI.TargetPosition := #Ax.AxisCtrl.MoveAbsTarget;
       END_IF;

       // Target position exceeds MAX limit
       // 
       #LimitExceeds := "M_CmpGT"(Xa := #Ax.AxisCtrl.MoveAbsTarget, Xb := #COut.MaxPosition, MODULE := #Sts.AxisModulo);
       IF #LimitExceeds THEN
           #Ax.AxisCtrl.MoveAbsTarget := #COut.MaxPosition;
           #HMI.TargetPosition := #Ax.AxisCtrl.MoveAbsTarget;
       END_IF;

   END_IF;
END_REGION

REGION Network 32 (SCL): Check missing position to reach the target
   #Sts.MissingToTarget := "M_PosAMinusPosB"(PosA := #Ax.AxisCtrl.MoveAbsTarget, PosB := #Pers_Data.ActualPosition, MODULE := #Sts.AxisModulo);

   //  Missing position to reach the target ABS value
   //  
   #Sts.MissingToTarget_ABS := ABS(#Sts.MissingToTarget);
END_REGION

REGION Network 33 (SCL): Status axis in target position

   #TON_InTargetPosition(IN := ABS(#Sts.MissingToTarget) <= #Par.PosTolerance, PT:=#Par.DelayInPosition);

   #Sts.InTargetPosition := #TON_InTargetPosition.Q AND #Ax.AxisSts.Homed AND (#Ax.AxisSts.Positioned OR NOT #Ax.AxisCtrl.MoveAbsolute);
END_REGION

REGION Network 34 (SCL): Axis Control (Velocity / Acceleration / Deceleration / Jerk)

   #COut.MaxVelocity := MIN(IN1 := #TO_Ax.DynamicLimits.MaxVelocity, IN2 := #TO_Ax.DynamicLimits.Velocity);

   #Ctrl.Vel := 0.0;


   IF #Ctrl.Bwd_Man OR #Ctrl.Fwd_Man OR #Ctrl.MoveToPos_Man THEN


       #Ctrl.Acc := #Par.Man.Acc;
       #Ctrl.Dec := #Par.Man.Dec;
       #Ctrl.Jerk := #Par.Man.Jerk;



       IF #Ctrl.Bwd_Man THEN

           #Ctrl.Vel := #Par.Man.VelBwd;

       ELSIF #Ctrl.Fwd_Man AND #Ctrl.Man_HighSpeed  THEN
           #Ctrl.Vel := #Par.Man.VelFwdHigh;

       ELSIF #Ctrl.Fwd_Man OR #Ctrl.MoveToPos_Man  THEN

           #Ctrl.Vel := #Par.Man.VelFwdLow;
       END_IF;



   ELSIF #Ctrl.MoveToPos_Aut OR #Ctrl.Bwd_Aut OR #Ctrl.Fwd_Aut  THEN

       #Ctrl.Vel := #CIn.Manager.Vel;

       #Ctrl.Acc := #CIn.Manager.Acc;
       #Ctrl.Dec := #CIn.Manager.Dec;
       #Ctrl.Jerk := #CIn.Manager.Jerk;


   END_IF;




   // Dynamic limits
   // 

   #Ctrl.Vel := MIN(IN1:=#Ctrl.Vel, IN2 := #COut.MaxVelocity);

   #Ctrl.Acc :=    MIN (IN1:=#Ctrl.Acc, IN2:= #TO_Ax.DynamicLimits.MaxAcceleration);
   IF #Ctrl.Acc <= 0.0 THEN
       #Ctrl.Acc :=  #Par.Man.Acc;
   END_IF;

   #Ctrl.Dec :=    MIN (IN1:=#Ctrl.Dec, IN2:= #TO_Ax.DynamicLimits.MaxDeceleration);
   IF #Ctrl.Dec <= 0.0 THEN
       #Ctrl.Dec :=  #Par.Man.Dec;
   END_IF;

   IF  #Ctrl.Jerk > 0.0 THEN

       #Ctrl.Jerk :=   MIN (IN1:= #Ctrl.Jerk,IN2:= #TO_Ax.DynamicLimits.MaxJerk);
   ELSE
       #Ctrl.Jerk := 0.0;
   END_IF;






   // Velocity override
   // 

   #TO_Ax.Override.Velocity := 100.0;

   IF #CIn.VelocityOverride.Enable THEN
       #TO_Ax.Override.Velocity := #CIn.VelocityOverride.Value;
   END_IF;


   // SLS velocity limit
   // 
   IF #ZSI.Door_Opened AND #Ctrl.Vel > #Config.SLS_VEL THEN
       #Ctrl.Vel := MIN(IN1:= #Ctrl.Vel, IN2:= #Config.SLS_VEL);
   END_IF;


   // Brake not open... Velocity  = 0.0
   // 
   IF #Config.Brake_Presence AND NOT #DataIn.Brake_M_Feedback THEN
       #Ctrl.Vel := 0.0;
   END_IF;

   // Init cycle force velocity = 0.0
   //
   IF #WritePar.Running OR #EncoderSelection.Running OR #ReloadPosition.Running OR #LoadPosition.Running  THEN
       #Ctrl.Vel := 0.0;
   END_IF;



   // Write dynamics value

   #Ax.AxisCtrl.Velocity :=   #Ctrl.Vel;
   #Ax.AxisCtrl.Acceleration := #Ctrl.Acc;
   #Ax.AxisCtrl.Deceleration := #Ctrl.Dec;
   #Ax.AxisCtrl.Jerk:=  #Ctrl.Jerk;
END_REGION

REGION Network 35 (SCL): Axis Control (Home Parameters) / Velocity & Dynamics
   #Ax.AxisCtrl.HomeMode := #Config.Ax.HomeMode;

   IF #ReloadPosition.Running THEN
       #Ax.AxisCtrl.HomePosition := #ReloadPosition.Ctrl_ReloadPosAx;
   ELSIF #LoadPosition.Running THEN
       #Ax.AxisCtrl.HomePosition := #LoadPosition.Ctrl_LoadPosAx;
   END_IF;
END_REGION

REGION Network 36: Move request in bwd / fwd direction case positioning
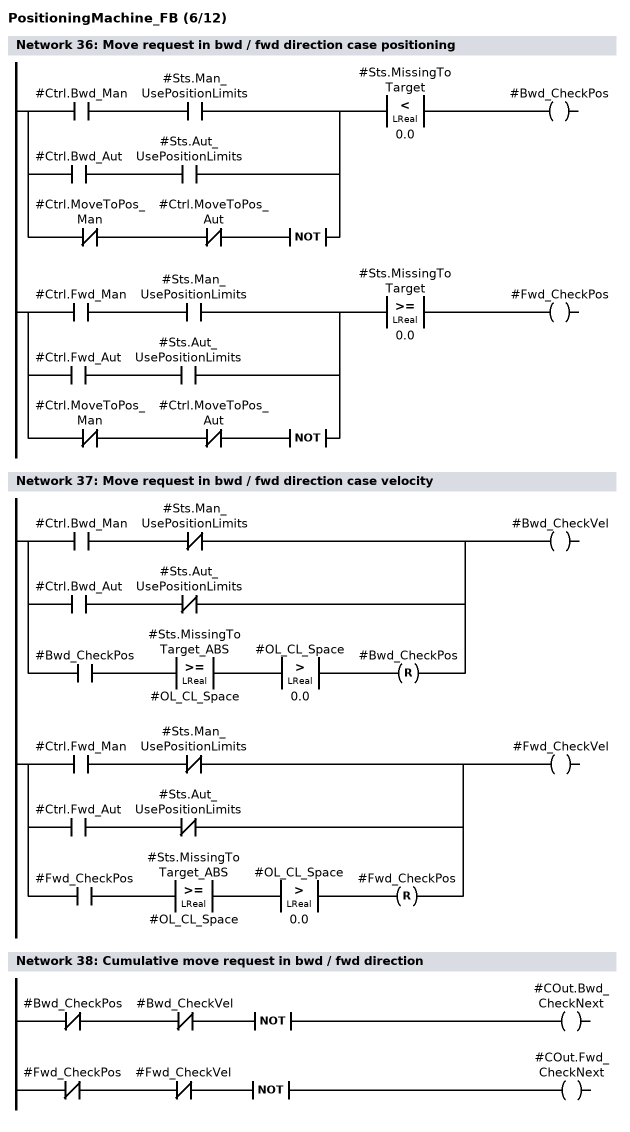
   RUNG wire#powerrail
      Contact( #Ctrl.Bwd_Man )
      Contact( #Sts.Man_UsePositionLimits )
      wire#w1
      { S7_Templates := "SrcType := LReal" } LT_Contact(in1 := #Sts.MissingToTarget, in2 := 0.0)
      Coil( #Bwd_CheckPos )
   END_RUNG
   RUNG wire#powerrail
      Contact( #Ctrl.Bwd_Aut )
      Contact( #Sts.Aut_UsePositionLimits )
   END_RUNG wire#w1
   RUNG wire#powerrail
      I_Contact( #Ctrl.MoveToPos_Man )
      I_Contact( #Ctrl.MoveToPos_Aut )
      Not()
   END_RUNG wire#w1
   RUNG wire#powerrail
      Contact( #Ctrl.Fwd_Man )
      Contact( #Sts.Man_UsePositionLimits )
      wire#w2
      { S7_Templates := "SrcType := LReal" } GE_Contact(in1 := #Sts.MissingToTarget, in2 := 0.0)
      Coil( #Fwd_CheckPos )
   END_RUNG
   RUNG wire#powerrail
      Contact( #Ctrl.Fwd_Aut )
      Contact( #Sts.Aut_UsePositionLimits )
   END_RUNG wire#w2
   RUNG wire#powerrail
      I_Contact( #Ctrl.MoveToPos_Man )
      I_Contact( #Ctrl.MoveToPos_Aut )
      Not()
   END_RUNG wire#w2
   // the same network as SCL:
   #Bwd_CheckPos := ((#Ctrl.Bwd_Man AND #Sts.Man_UsePositionLimits) OR (#Ctrl.Bwd_Aut AND #Sts.Aut_UsePositionLimits) OR NOT (NOT #Ctrl.MoveToPos_Man AND NOT #Ctrl.MoveToPos_Aut)) AND (#Sts.MissingToTarget < 0.0);
   #Fwd_CheckPos := ((#Ctrl.Fwd_Man AND #Sts.Man_UsePositionLimits) OR (#Ctrl.Fwd_Aut AND #Sts.Aut_UsePositionLimits) OR NOT (NOT #Ctrl.MoveToPos_Man AND NOT #Ctrl.MoveToPos_Aut)) AND (#Sts.MissingToTarget >= 0.0);
END_REGION

REGION Network 37: Move request in bwd / fwd direction case velocity
   RUNG wire#powerrail
      Contact( #Ctrl.Bwd_Man )
      I_Contact( #Sts.Man_UsePositionLimits )
      wire#w1
      Coil( #Bwd_CheckVel )
   END_RUNG
   RUNG wire#powerrail
      Contact( #Ctrl.Bwd_Aut )
      I_Contact( #Sts.Aut_UsePositionLimits )
   END_RUNG wire#w1
   RUNG wire#powerrail
      Contact( #Bwd_CheckPos )
      { S7_Templates := "SrcType := LReal" } GE_Contact(in1 := #Sts.MissingToTarget_ABS, in2 := #OL_CL_Space)
      { S7_Templates := "SrcType := LReal" } GT_Contact(in1 := #OL_CL_Space, in2 := 0.0)
      R_Coil( #Bwd_CheckPos )
   END_RUNG wire#w1
   RUNG wire#powerrail
      Contact( #Ctrl.Fwd_Man )
      I_Contact( #Sts.Man_UsePositionLimits )
      wire#w2
      Coil( #Fwd_CheckVel )
   END_RUNG
   RUNG wire#powerrail
      Contact( #Ctrl.Fwd_Aut )
      I_Contact( #Sts.Aut_UsePositionLimits )
   END_RUNG wire#w2
   RUNG wire#powerrail
      Contact( #Fwd_CheckPos )
      { S7_Templates := "SrcType := LReal" } GE_Contact(in1 := #Sts.MissingToTarget_ABS, in2 := #OL_CL_Space)
      { S7_Templates := "SrcType := LReal" } GT_Contact(in1 := #OL_CL_Space, in2 := 0.0)
      R_Coil( #Fwd_CheckPos )
   END_RUNG wire#w2
   // the same network as SCL:
   #_w1 := #Bwd_CheckPos AND (#Sts.MissingToTarget_ABS >= #OL_CL_Space) AND (#OL_CL_Space > 0.0);
   IF #_w1 THEN #Bwd_CheckPos := FALSE; END_IF;
   #Bwd_CheckVel := (#Ctrl.Bwd_Man AND NOT #Sts.Man_UsePositionLimits) OR (#Ctrl.Bwd_Aut AND NOT #Sts.Aut_UsePositionLimits) OR #_w1;
   #_w2 := #Fwd_CheckPos AND (#Sts.MissingToTarget_ABS >= #OL_CL_Space) AND (#OL_CL_Space > 0.0);
   IF #_w2 THEN #Fwd_CheckPos := FALSE; END_IF;
   #Fwd_CheckVel := (#Ctrl.Fwd_Man AND NOT #Sts.Man_UsePositionLimits) OR (#Ctrl.Fwd_Aut AND NOT #Sts.Aut_UsePositionLimits) OR #_w2;
END_REGION

REGION Network 38: Cumulative move request in bwd / fwd direction
   RUNG wire#powerrail
      I_Contact( #Bwd_CheckPos )
      I_Contact( #Bwd_CheckVel )
      Not()
      Coil( #COut.Bwd_CheckNext )
   END_RUNG
   RUNG wire#powerrail
      I_Contact( #Fwd_CheckPos )
      I_Contact( #Fwd_CheckVel )
      Not()
      Coil( #COut.Fwd_CheckNext )
   END_RUNG
   // the same network as SCL:
   #COut.Bwd_CheckNext := NOT (NOT #Bwd_CheckPos AND NOT #Bwd_CheckVel);
   #COut.Fwd_CheckNext := NOT (NOT #Fwd_CheckPos AND NOT #Fwd_CheckVel);
END_REGION

REGION Network 39: Conditions
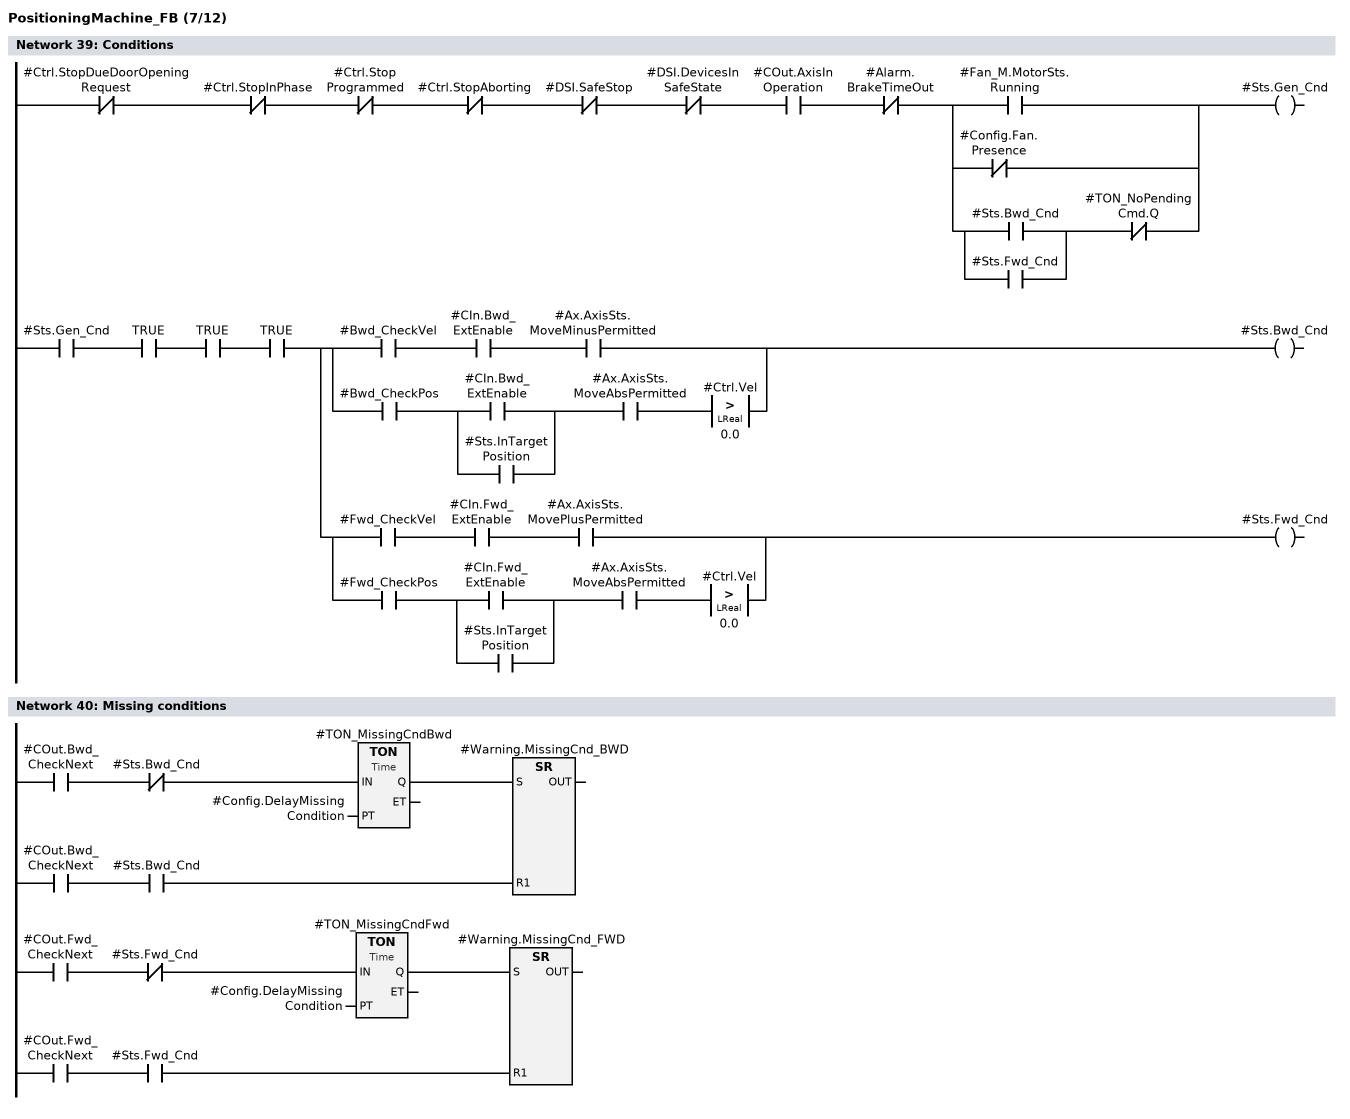
   RUNG wire#powerrail
      I_Contact( #Ctrl.StopDueDoorOpeningRequest )
      I_Contact( #Ctrl.StopInPhase )
      I_Contact( #Ctrl.StopProgrammed )
      I_Contact( #Ctrl.StopAborting )
      I_Contact( #DSI.SafeStop )
      I_Contact( #DSI.DevicesInSafeState )
      Contact( #COut.AxisInOperation )
      I_Contact( #Alarm.BrakeTimeOut )
      wire#w1
      Contact( #Fan_M.MotorSts.Running )
      wire#w2
      Coil( #Sts.Gen_Cnd )
   END_RUNG
   RUNG wire#w1
      I_Contact( #Config.Fan.Presence )
   END_RUNG wire#w2
   RUNG wire#w1
      Contact( #Sts.Bwd_Cnd )
      wire#w3
      I_Contact( #TON_NoPendingCmd.Q )
   END_RUNG wire#w2
   RUNG wire#w1
      Contact( #Sts.Fwd_Cnd )
   END_RUNG wire#w3
   RUNG wire#powerrail
      Contact( #Sts.Gen_Cnd )
      Contact( TRUE )
      Contact( TRUE )
      Contact( TRUE )
      wire#w4
      Contact( #Bwd_CheckVel )
      Contact( #CIn.Bwd_ExtEnable )
      Contact( #Ax.AxisSts.MoveMinusPermitted )
      wire#w5
      Coil( #Sts.Bwd_Cnd )
   END_RUNG
   RUNG wire#w4
      Contact( #Bwd_CheckPos )
      wire#w6
      Contact( #CIn.Bwd_ExtEnable )
      wire#w7
      Contact( #Ax.AxisSts.MoveAbsPermitted )
      { S7_Templates := "SrcType := LReal" } GT_Contact(in1 := #Ctrl.Vel, in2 := 0.0)
   END_RUNG wire#w5
   RUNG wire#w6
      Contact( #Sts.InTargetPosition )
   END_RUNG wire#w7
   RUNG wire#w4
      Contact( #Fwd_CheckVel )
      Contact( #CIn.Fwd_ExtEnable )
      Contact( #Ax.AxisSts.MovePlusPermitted )
      wire#w8
      Coil( #Sts.Fwd_Cnd )
   END_RUNG
   RUNG wire#w4
      Contact( #Fwd_CheckPos )
      wire#w9
      Contact( #CIn.Fwd_ExtEnable )
      wire#w10
      Contact( #Ax.AxisSts.MoveAbsPermitted )
      { S7_Templates := "SrcType := LReal" } GT_Contact(in1 := #Ctrl.Vel, in2 := 0.0)
   END_RUNG wire#w8
   RUNG wire#w9
      Contact( #Sts.InTargetPosition )
   END_RUNG wire#w10
   // the same network as SCL:
   #Sts.Gen_Cnd := NOT #Ctrl.StopDueDoorOpeningRequest AND NOT #Ctrl.StopInPhase AND NOT #Ctrl.StopProgrammed AND NOT #Ctrl.StopAborting AND NOT #DSI.SafeStop AND NOT #DSI.DevicesInSafeState AND #COut.AxisInOperation AND NOT #Alarm.BrakeTimeOut AND (#Fan_M.MotorSts.Running OR NOT #Config.Fan.Presence OR ((#Sts.Bwd_Cnd OR #Sts.Fwd_Cnd) AND NOT #TON_NoPendingCmd.Q));
   #_w1 := #Sts.Gen_Cnd AND TRUE AND TRUE AND TRUE;
   #Sts.Bwd_Cnd := #_w1 AND ((#Bwd_CheckVel AND #CIn.Bwd_ExtEnable AND #Ax.AxisSts.MoveMinusPermitted) OR (#Bwd_CheckPos AND (#CIn.Bwd_ExtEnable OR #Sts.InTargetPosition) AND #Ax.AxisSts.MoveAbsPermitted AND (#Ctrl.Vel > 0.0)));
   #Sts.Fwd_Cnd := #_w1 AND ((#Fwd_CheckVel AND #CIn.Fwd_ExtEnable AND #Ax.AxisSts.MovePlusPermitted) OR (#Fwd_CheckPos AND (#CIn.Fwd_ExtEnable OR #Sts.InTargetPosition) AND #Ax.AxisSts.MoveAbsPermitted AND (#Ctrl.Vel > 0.0)));
END_REGION

REGION Network 40: Missing conditions
   RUNG wire#powerrail
      Contact( #COut.Bwd_CheckNext )
      I_Contact( #Sts.Bwd_Cnd )
      { S7_Templates := "time_type := Time" } #TON_MissingCndBwd.TON(pt := #Config.DelayMissingCondition, et =>)
      S_SR(operand := #Warning.MissingCnd_BWD, r1 := wire#w1)
   END_RUNG
   RUNG wire#powerrail
      Contact( #COut.Bwd_CheckNext )
      Contact( #Sts.Bwd_Cnd )
   END_RUNG wire#w1
   RUNG wire#powerrail
      Contact( #COut.Fwd_CheckNext )
      I_Contact( #Sts.Fwd_Cnd )
      { S7_Templates := "time_type := Time" } #TON_MissingCndFwd.TON(pt := #Config.DelayMissingCondition, et =>)
      S_SR(operand := #Warning.MissingCnd_FWD, r1 := wire#w2)
   END_RUNG
   RUNG wire#powerrail
      Contact( #COut.Fwd_CheckNext )
      Contact( #Sts.Fwd_Cnd )
   END_RUNG wire#w2
   // the same network as SCL:
   #TON_MissingCndBwd(IN := #COut.Bwd_CheckNext AND NOT #Sts.Bwd_Cnd, PT := #Config.DelayMissingCondition);   // TON
   IF #TON_MissingCndBwd.Q THEN
       #Warning.MissingCnd_BWD := TRUE;   // SR flip-flop
   END_IF;
   IF #COut.Bwd_CheckNext AND #Sts.Bwd_Cnd THEN #Warning.MissingCnd_BWD := FALSE; END_IF;
   #TON_MissingCndFwd(IN := #COut.Fwd_CheckNext AND NOT #Sts.Fwd_Cnd, PT := #Config.DelayMissingCondition);   // TON
   IF #TON_MissingCndFwd.Q THEN
       #Warning.MissingCnd_FWD := TRUE;   // SR flip-flop
   END_IF;
   IF #COut.Fwd_CheckNext AND #Sts.Fwd_Cnd THEN #Warning.MissingCnd_FWD := FALSE; END_IF;
END_REGION

REGION Network 41: Axis Control (bit)
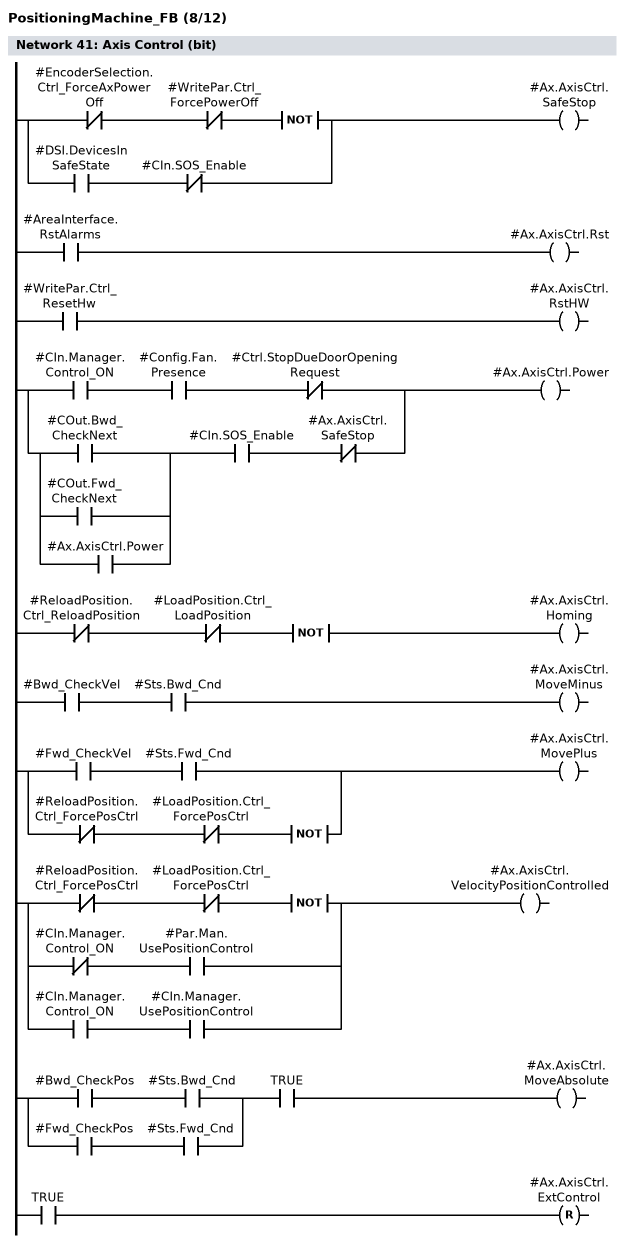
   RUNG wire#powerrail
      I_Contact( #EncoderSelection.Ctrl_ForceAxPowerOff )
      I_Contact( #WritePar.Ctrl_ForcePowerOff )
      Not()
      wire#w1
      Coil( #Ax.AxisCtrl.SafeStop )
   END_RUNG
   RUNG wire#powerrail
      Contact( #DSI.DevicesInSafeState )
      I_Contact( #CIn.SOS_Enable )
   END_RUNG wire#w1
   RUNG wire#powerrail
      Contact( #AreaInterface.RstAlarms )
      Coil( #Ax.AxisCtrl.Rst )
   END_RUNG
   RUNG wire#powerrail
      Contact( #WritePar.Ctrl_ResetHw )
      Coil( #Ax.AxisCtrl.RstHW )
   END_RUNG
   RUNG wire#powerrail
      Contact( #CIn.Manager.Control_ON )
      Contact( #Config.Fan.Presence )
      I_Contact( #Ctrl.StopDueDoorOpeningRequest )
      wire#w2
      Coil( #Ax.AxisCtrl.Power )
   END_RUNG
   RUNG wire#powerrail
      Contact( #COut.Bwd_CheckNext )
      wire#w3
      Contact( #CIn.SOS_Enable )
      I_Contact( #Ax.AxisCtrl.SafeStop )
   END_RUNG wire#w2
   RUNG wire#powerrail
      Contact( #COut.Fwd_CheckNext )
   END_RUNG wire#w3
   RUNG wire#powerrail
      Contact( #Ax.AxisCtrl.Power )
   END_RUNG wire#w3
   RUNG wire#powerrail
      I_Contact( #ReloadPosition.Ctrl_ReloadPosition )
      I_Contact( #LoadPosition.Ctrl_LoadPosition )
      Not()
      Coil( #Ax.AxisCtrl.Homing )
   END_RUNG
   RUNG wire#powerrail
      Contact( #Bwd_CheckVel )
      Contact( #Sts.Bwd_Cnd )
      Coil( #Ax.AxisCtrl.MoveMinus )
   END_RUNG
   RUNG wire#powerrail
      Contact( #Fwd_CheckVel )
      Contact( #Sts.Fwd_Cnd )
      wire#w4
      Coil( #Ax.AxisCtrl.MovePlus )
   END_RUNG
   RUNG wire#powerrail
      I_Contact( #ReloadPosition.Ctrl_ForcePosCtrl )
      I_Contact( #LoadPosition.Ctrl_ForcePosCtrl )
      Not()
   END_RUNG wire#w4
   RUNG wire#powerrail
      I_Contact( #ReloadPosition.Ctrl_ForcePosCtrl )
      I_Contact( #LoadPosition.Ctrl_ForcePosCtrl )
      Not()
      wire#w5
      Coil( #Ax.AxisCtrl.VelocityPositionControlled )
   END_RUNG
   RUNG wire#powerrail
      I_Contact( #CIn.Manager.Control_ON )
      Contact( #Par.Man.UsePositionControl )
   END_RUNG wire#w5
   RUNG wire#powerrail
      Contact( #CIn.Manager.Control_ON )
      Contact( #CIn.Manager.UsePositionControl )
   END_RUNG wire#w5
   RUNG wire#powerrail
      Contact( #Bwd_CheckPos )
      Contact( #Sts.Bwd_Cnd )
      wire#w6
      Contact( TRUE )
      Coil( #Ax.AxisCtrl.MoveAbsolute )
   END_RUNG
   RUNG wire#powerrail
      Contact( #Fwd_CheckPos )
      Contact( #Sts.Fwd_Cnd )
   END_RUNG wire#w6
   RUNG wire#powerrail
      Contact( TRUE )
      R_Coil( #Ax.AxisCtrl.ExtControl )
   END_RUNG
   // the same network as SCL:
   #Ax.AxisCtrl.SafeStop := NOT (NOT #EncoderSelection.Ctrl_ForceAxPowerOff AND NOT #WritePar.Ctrl_ForcePowerOff) OR (#DSI.DevicesInSafeState AND NOT #CIn.SOS_Enable);
   #Ax.AxisCtrl.Rst := #AreaInterface.RstAlarms;
   #Ax.AxisCtrl.RstHW := #WritePar.Ctrl_ResetHw;
   #Ax.AxisCtrl.Power := (#CIn.Manager.Control_ON AND #Config.Fan.Presence AND NOT #Ctrl.StopDueDoorOpeningRequest) OR ((#COut.Bwd_CheckNext OR #COut.Fwd_CheckNext OR #Ax.AxisCtrl.Power) AND #CIn.SOS_Enable AND NOT #Ax.AxisCtrl.SafeStop);
   #Ax.AxisCtrl.Homing := NOT (NOT #ReloadPosition.Ctrl_ReloadPosition AND NOT #LoadPosition.Ctrl_LoadPosition);
   #Ax.AxisCtrl.MoveMinus := #Bwd_CheckVel AND #Sts.Bwd_Cnd;
   #Ax.AxisCtrl.MovePlus := (#Fwd_CheckVel AND #Sts.Fwd_Cnd) OR NOT (NOT #ReloadPosition.Ctrl_ForcePosCtrl AND NOT #LoadPosition.Ctrl_ForcePosCtrl);
   #Ax.AxisCtrl.VelocityPositionControlled := NOT (NOT #ReloadPosition.Ctrl_ForcePosCtrl AND NOT #LoadPosition.Ctrl_ForcePosCtrl) OR (NOT #CIn.Manager.Control_ON AND #Par.Man.UsePositionControl) OR (#CIn.Manager.Control_ON AND #CIn.Manager.UsePositionControl);
   #Ax.AxisCtrl.MoveAbsolute := ((#Bwd_CheckPos AND #Sts.Bwd_Cnd) OR (#Fwd_CheckPos AND #Sts.Fwd_Cnd)) AND TRUE;
   IF TRUE THEN #Ax.AxisCtrl.ExtControl := FALSE; END_IF;
END_REGION

REGION Network 42: Axis manager
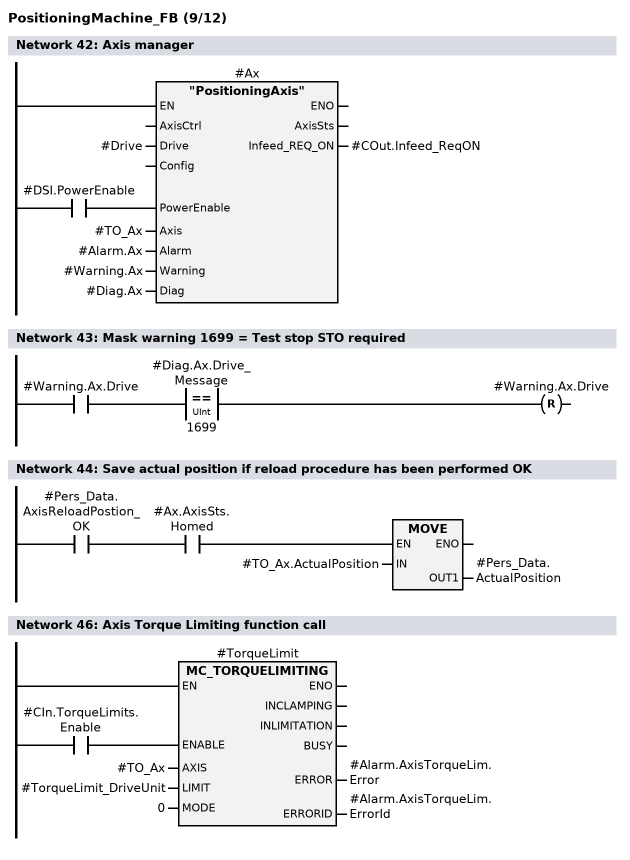
   RUNG wire#powerrail
      #Ax(PowerEnable := wire#w1, AxisCtrl :=, Drive := #Drive, Config :=, Axis := #TO_Ax, Alarm := #Alarm.Ax, Warning := #Warning.Ax, Diag := #Diag.Ax, AxisSts =>, Infeed_REQ_ON => #COut.Infeed_ReqON)
   END_RUNG
   RUNG wire#powerrail
      Contact( #DSI.PowerEnable )
   END_RUNG wire#w1
   // the same network as SCL:
   #Ax(Drive := #Drive,   // "PositioningAxis"
       PowerEnable := #DSI.PowerEnable,
       Axis := #TO_Ax,
       Alarm := #Alarm.Ax,
       Warning := #Warning.Ax,
       Diag := #Diag.Ax,
       Infeed_REQ_ON => #COut.Infeed_ReqON);
END_REGION

REGION Network 43: Mask warning 1699 = Test stop STO required
   RUNG wire#powerrail
      Contact( #Warning.Ax.Drive )
      { S7_Templates := "SrcType := UInt" } EQ_Contact(in1 := #Diag.Ax.Drive_Message, in2 := 1699)
      R_Coil( #Warning.Ax.Drive )
   END_RUNG
   // the same network as SCL:
   IF #Warning.Ax.Drive AND (#Diag.Ax.Drive_Message = 1699) THEN #Warning.Ax.Drive := FALSE; END_IF;
END_REGION

REGION Network 44: Save actual position if reload procedure has been performed OK
   RUNG wire#powerrail
      Contact( #Pers_Data.AxisReloadPostion_OK )
      Contact( #Ax.AxisSts.Homed )
      { S7_GenerateENO := "TRUE" } Move(in := #TO_Ax.ActualPosition, out1 => #Pers_Data.ActualPosition)
   END_RUNG
   // the same network as SCL:
   IF #Pers_Data.AxisReloadPostion_OK AND #Ax.AxisSts.Homed THEN
       #Pers_Data.ActualPosition := #TO_Ax.ActualPosition;
   END_IF;
END_REGION

REGION Network 45 (SCL): Axis Torque Limit normalization

   #TorqueLimit_EngUnit := LIMIT(MN:=0.0, IN:=#CIn.TorqueLimits.Value, MX:=(#TO_Ax.Actor.DriveParameter.ReferenceTorque / 2.0));

   #TorqueLimit_Percentage := #TorqueLimit_EngUnit / (#TO_Ax.Actor.DriveParameter.ReferenceTorque / 2.0)  * 100.0;

   #TorqueLimit_DriveUnit := 30720 / 100.0 * #TorqueLimit_Percentage;



   #TorqueLimit_DriveUnit := #TorqueLimit_Percentage;
END_REGION

REGION Network 46: Axis Torque Limiting function call
   RUNG wire#powerrail
      #TorqueLimit.MC_TORQUELIMITING(Enable := wire#w1, Axis := #TO_Ax, Limit := #TorqueLimit_DriveUnit, Mode := 0, InClamping =>, InLimitation =>, Busy =>, Error => #Alarm.AxisTorqueLim.Error, ErrorId => #Alarm.AxisTorqueLim.ErrorId)
   END_RUNG
   RUNG wire#powerrail
      Contact( #CIn.TorqueLimits.Enable )
   END_RUNG wire#w1
   // the same network as SCL:
   #TorqueLimit(Enable := #CIn.TorqueLimits.Enable,   // MC_TORQUELIMITING
                Axis := #TO_Ax,
                Limit := #TorqueLimit_DriveUnit,
                Mode := 0,
                Error => #Alarm.AxisTorqueLim.Error,
                ErrorId => #Alarm.AxisTorqueLim.ErrorId);
END_REGION

REGION Network 47: Coordination Out
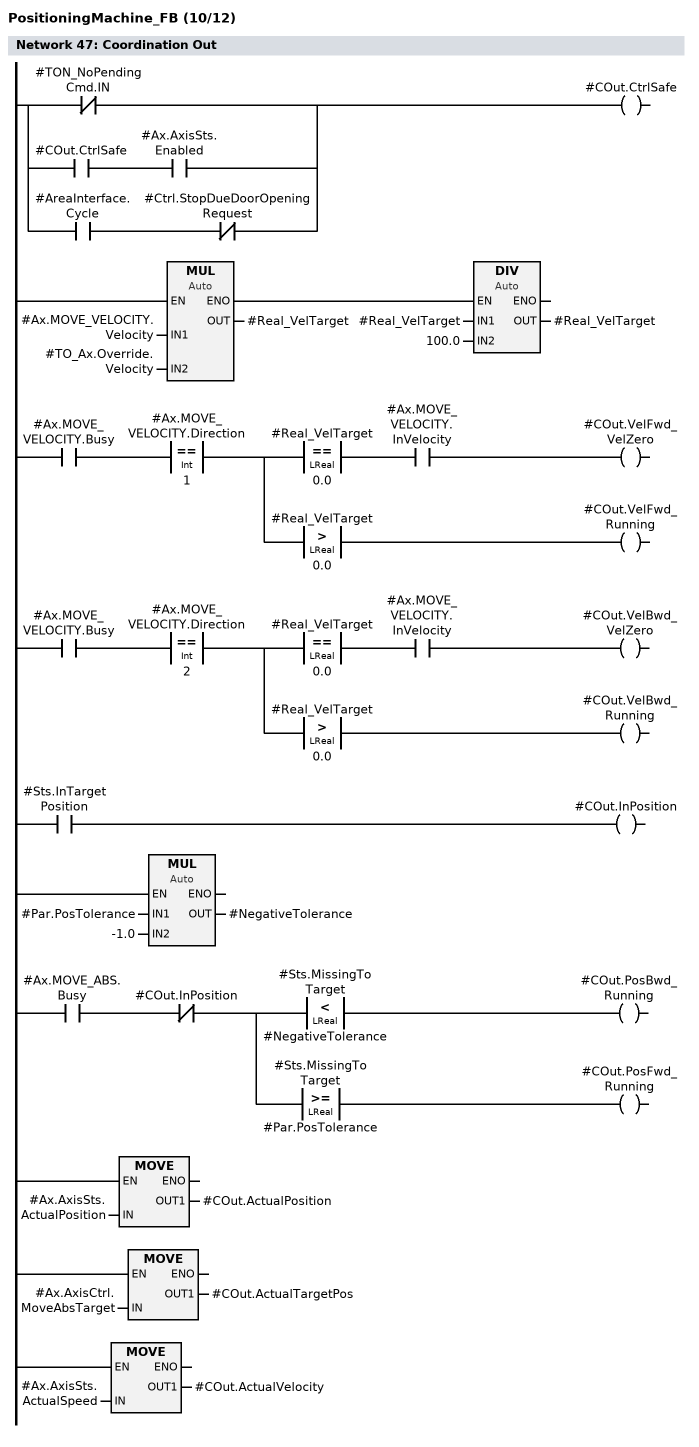
   RUNG wire#powerrail
      I_Contact( #TON_NoPendingCmd.IN )
      wire#w1
      Coil( #COut.CtrlSafe )
   END_RUNG
   RUNG wire#powerrail
      Contact( #COut.CtrlSafe )
      Contact( #Ax.AxisSts.Enabled )
   END_RUNG wire#w1
   RUNG wire#powerrail
      Contact( #AreaInterface.Cycle )
      I_Contact( #Ctrl.StopDueDoorOpeningRequest )
   END_RUNG wire#w1
   RUNG wire#powerrail
      { S7_GenerateENO := "TRUE" } Mul(in1 := #Ax.MOVE_VELOCITY.Velocity, in2 := #TO_Ax.Override.Velocity, out => #Real_VelTarget)
      { S7_GenerateENO := "TRUE" } Div(in1 := #Real_VelTarget, in2 := 100.0, out => #Real_VelTarget)
   END_RUNG
   RUNG wire#powerrail
      Contact( #Ax.MOVE_VELOCITY.Busy )
      { S7_Templates := "SrcType := Int" } EQ_Contact(in1 := #Ax.MOVE_VELOCITY.Direction, in2 := 1)
      wire#w2
      { S7_Templates := "SrcType := LReal" } EQ_Contact(in1 := #Real_VelTarget, in2 := 0.0)
      Contact( #Ax.MOVE_VELOCITY.InVelocity )
      Coil( #COut.VelFwd_VelZero )
   END_RUNG
   RUNG wire#w2
      { S7_Templates := "SrcType := LReal" } GT_Contact(in1 := #Real_VelTarget, in2 := 0.0)
      Coil( #COut.VelFwd_Running )
   END_RUNG
   RUNG wire#powerrail
      Contact( #Ax.MOVE_VELOCITY.Busy )
      { S7_Templates := "SrcType := Int" } EQ_Contact(in1 := #Ax.MOVE_VELOCITY.Direction, in2 := 2)
      wire#w3
      { S7_Templates := "SrcType := LReal" } EQ_Contact(in1 := #Real_VelTarget, in2 := 0.0)
      Contact( #Ax.MOVE_VELOCITY.InVelocity )
      Coil( #COut.VelBwd_VelZero )
   END_RUNG
   RUNG wire#w3
      { S7_Templates := "SrcType := LReal" } GT_Contact(in1 := #Real_VelTarget, in2 := 0.0)
      Coil( #COut.VelBwd_Running )
   END_RUNG
   RUNG wire#powerrail
      Contact( #Sts.InTargetPosition )
      Coil( #COut.InPosition )
   END_RUNG
   RUNG wire#powerrail
      Mul(in1 := #Par.PosTolerance, in2 := -1.0, out => #NegativeTolerance)
   END_RUNG
   RUNG wire#powerrail
      Contact( #Ax.MOVE_ABS.Busy )
      I_Contact( #COut.InPosition )
      wire#w4
      { S7_Templates := "SrcType := LReal" } LT_Contact(in1 := #Sts.MissingToTarget, in2 := #NegativeTolerance)
      Coil( #COut.PosBwd_Running )
   END_RUNG
   RUNG wire#w4
      { S7_Templates := "SrcType := LReal" } GE_Contact(in1 := #Sts.MissingToTarget, in2 := #Par.PosTolerance)
      Coil( #COut.PosFwd_Running )
   END_RUNG
   RUNG wire#powerrail
      Move(in := #Ax.AxisSts.ActualPosition, out1 => #COut.ActualPosition)
   END_RUNG
   RUNG wire#powerrail
      Move(in := #Ax.AxisCtrl.MoveAbsTarget, out1 => #COut.ActualTargetPos)
   END_RUNG
   RUNG wire#powerrail
      Move(in := #Ax.AxisSts.ActualSpeed, out1 => #COut.ActualVelocity)
   END_RUNG
   // the same network as SCL:
   // ENO of a box is taken as its EN; it also drops when the box reports an error
   #COut.CtrlSafe := NOT #TON_NoPendingCmd.IN OR (#COut.CtrlSafe AND #Ax.AxisSts.Enabled) OR (#AreaInterface.Cycle AND NOT #Ctrl.StopDueDoorOpeningRequest);
   #Real_VelTarget := #Ax.MOVE_VELOCITY.Velocity * #TO_Ax.Override.Velocity;
   #Real_VelTarget := #Real_VelTarget / 100.0;
   #_w1 := #Ax.MOVE_VELOCITY.Busy AND (#Ax.MOVE_VELOCITY.Direction = 1);
   #COut.VelFwd_VelZero := #_w1 AND (#Real_VelTarget = 0.0) AND #Ax.MOVE_VELOCITY.InVelocity;
   #COut.VelFwd_Running := #_w1 AND (#Real_VelTarget > 0.0);
   #_w2 := #Ax.MOVE_VELOCITY.Busy AND (#Ax.MOVE_VELOCITY.Direction = 2);
   #COut.VelBwd_VelZero := #_w2 AND (#Real_VelTarget = 0.0) AND #Ax.MOVE_VELOCITY.InVelocity;
   #COut.VelBwd_Running := #_w2 AND (#Real_VelTarget > 0.0);
   #COut.InPosition := #Sts.InTargetPosition;
   #NegativeTolerance := #Par.PosTolerance * (-1.0);
   #_w3 := #Ax.MOVE_ABS.Busy AND NOT #COut.InPosition;
   #COut.PosBwd_Running := #_w3 AND (#Sts.MissingToTarget < #NegativeTolerance);
   #COut.PosFwd_Running := #_w3 AND (#Sts.MissingToTarget >= #Par.PosTolerance);
   #COut.ActualPosition := #Ax.AxisSts.ActualPosition;
   #COut.ActualTargetPos := #Ax.AxisCtrl.MoveAbsTarget;
   #COut.ActualVelocity := #Ax.AxisSts.ActualSpeed;
END_REGION

REGION Network 48: >
END_REGION

REGION Network 49: <<< MOTOR FAN >>>
END_REGION

REGION Network 50: Run
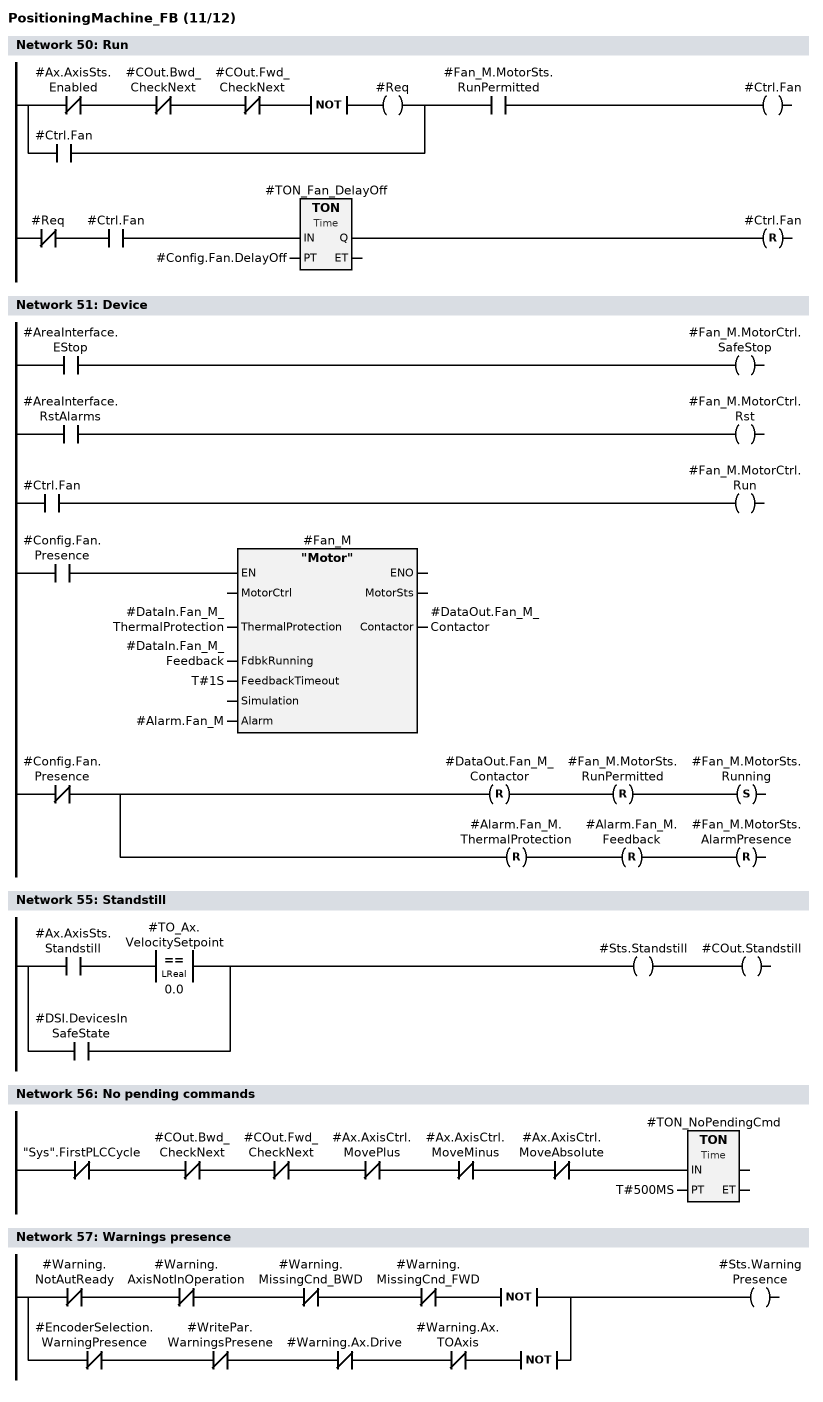
   RUNG wire#powerrail
      I_Contact( #Ax.AxisSts.Enabled )
      I_Contact( #COut.Bwd_CheckNext )
      I_Contact( #COut.Fwd_CheckNext )
      Not()
      Coil( #Req )
      wire#w1
      Contact( #Fan_M.MotorSts.RunPermitted )
      Coil( #Ctrl.Fan )
   END_RUNG
   RUNG wire#powerrail
      Contact( #Ctrl.Fan )
   END_RUNG wire#w1
   RUNG wire#powerrail
      I_Contact( #Req )
      Contact( #Ctrl.Fan )
      { S7_Templates := "time_type := Time" } #TON_Fan_DelayOff.TON(pt := #Config.Fan.DelayOff, et =>)
      R_Coil( #Ctrl.Fan )
   END_RUNG
   // the same network as SCL:
   #Req := NOT (NOT #Ax.AxisSts.Enabled AND NOT #COut.Bwd_CheckNext AND NOT #COut.Fwd_CheckNext);
   #Ctrl.Fan := (#Req OR #Ctrl.Fan) AND #Fan_M.MotorSts.RunPermitted;
   #TON_Fan_DelayOff(IN := NOT #Req AND #Ctrl.Fan, PT := #Config.Fan.DelayOff);   // TON
   IF #TON_Fan_DelayOff.Q THEN #Ctrl.Fan := FALSE; END_IF;
END_REGION

REGION Network 51: Device
   RUNG wire#powerrail
      Contact( #AreaInterface.EStop )
      Coil( #Fan_M.MotorCtrl.SafeStop )
   END_RUNG
   RUNG wire#powerrail
      Contact( #AreaInterface.RstAlarms )
      Coil( #Fan_M.MotorCtrl.Rst )
   END_RUNG
   RUNG wire#powerrail
      Contact( #Ctrl.Fan )
      Coil( #Fan_M.MotorCtrl.Run )
   END_RUNG
   RUNG wire#powerrail
      Contact( #Config.Fan.Presence )
      #Fan_M(MotorCtrl :=, ThermalProtection := #DataIn.Fan_M_ThermalProtection, FdbkRunning := #DataIn.Fan_M_Feedback, FeedbackTimeout := T#1S, Simulation :=, Alarm := #Alarm.Fan_M, MotorSts =>, Contactor => #DataOut.Fan_M_Contactor)
   END_RUNG
   RUNG wire#powerrail
      I_Contact( #Config.Fan.Presence )
      wire#w1
      R_Coil( #DataOut.Fan_M_Contactor )
      R_Coil( #Fan_M.MotorSts.RunPermitted )
      S_Coil( #Fan_M.MotorSts.Running )
   END_RUNG
   RUNG wire#w1
      R_Coil( #Alarm.Fan_M.ThermalProtection )
      R_Coil( #Alarm.Fan_M.Feedback )
      R_Coil( #Fan_M.MotorSts.AlarmPresence )
   END_RUNG
   // the same network as SCL:
   #Fan_M.MotorCtrl.SafeStop := #AreaInterface.EStop;
   #Fan_M.MotorCtrl.Rst := #AreaInterface.RstAlarms;
   #Fan_M.MotorCtrl.Run := #Ctrl.Fan;
   IF #Config.Fan.Presence THEN
       #Fan_M(ThermalProtection := #DataIn.Fan_M_ThermalProtection,   // "Motor"
              FdbkRunning := #DataIn.Fan_M_Feedback,
              FeedbackTimeout := T#1S,
              Alarm := #Alarm.Fan_M,
              Contactor => #DataOut.Fan_M_Contactor);
   END_IF;
   IF NOT #Config.Fan.Presence THEN
       #DataOut.Fan_M_Contactor := FALSE;
       #Fan_M.MotorSts.RunPermitted := FALSE;
       #Fan_M.MotorSts.Running := TRUE;
       #Alarm.Fan_M.ThermalProtection := FALSE;
       #Alarm.Fan_M.Feedback := FALSE;
       #Fan_M.MotorSts.AlarmPresence := FALSE;
   END_IF;
END_REGION

REGION Network 52: >
END_REGION

REGION Network 53: >
END_REGION

REGION Network 54: <<< MACHINE STATUS >>>
END_REGION

REGION Network 55: Standstill
   RUNG wire#powerrail
      Contact( #Ax.AxisSts.Standstill )
      { S7_Templates := "SrcType := LReal" } EQ_Contact(in1 := #TO_Ax.VelocitySetpoint, in2 := 0.0)
      wire#w1
      Coil( #Sts.Standstill )
      Coil( #COut.Standstill )
   END_RUNG
   RUNG wire#powerrail
      Contact( #DSI.DevicesInSafeState )
   END_RUNG wire#w1
   // the same network as SCL:
   #Sts.Standstill := (#Ax.AxisSts.Standstill AND (#TO_Ax.VelocitySetpoint = 0.0)) OR #DSI.DevicesInSafeState;
   #COut.Standstill := #Sts.Standstill;
END_REGION

REGION Network 56: No pending commands
   RUNG wire#powerrail
      I_Contact( "Sys".FirstPLCCycle )
      I_Contact( #COut.Bwd_CheckNext )
      I_Contact( #COut.Fwd_CheckNext )
      I_Contact( #Ax.AxisCtrl.MovePlus )
      I_Contact( #Ax.AxisCtrl.MoveMinus )
      I_Contact( #Ax.AxisCtrl.MoveAbsolute )
      { S7_Templates := "time_type := Time" } #TON_NoPendingCmd.TON(pt := T#500MS, et =>)
   END_RUNG
   // the same network as SCL:
   #TON_NoPendingCmd(IN := NOT "Sys".FirstPLCCycle AND NOT #COut.Bwd_CheckNext AND NOT #COut.Fwd_CheckNext AND NOT #Ax.AxisCtrl.MovePlus AND NOT #Ax.AxisCtrl.MoveMinus AND NOT #Ax.AxisCtrl.MoveAbsolute,   // TON
                     PT := T#500MS);
END_REGION

REGION Network 57: Warnings presence
   RUNG wire#powerrail
      I_Contact( #Warning.NotAutReady )
      I_Contact( #Warning.AxisNotInOperation )
      I_Contact( #Warning.MissingCnd_BWD )
      I_Contact( #Warning.MissingCnd_FWD )
      Not()
      wire#w1
      Coil( #Sts.WarningPresence )
   END_RUNG
   RUNG wire#powerrail
      I_Contact( #EncoderSelection.WarningPresence )
      I_Contact( #WritePar.WarningsPresene )
      I_Contact( #Warning.Ax.Drive )
      I_Contact( #Warning.Ax.TOAxis )
      Not()
   END_RUNG wire#w1
   // the same network as SCL:
   #Sts.WarningPresence := NOT (NOT #Warning.NotAutReady AND NOT #Warning.AxisNotInOperation AND NOT #Warning.MissingCnd_BWD AND NOT #Warning.MissingCnd_FWD) OR NOT (NOT #EncoderSelection.WarningPresence AND NOT #WritePar.WarningsPresene AND NOT #Warning.Ax.Drive AND NOT #Warning.Ax.TOAxis);
END_REGION

REGION Network 58: Alarms presence
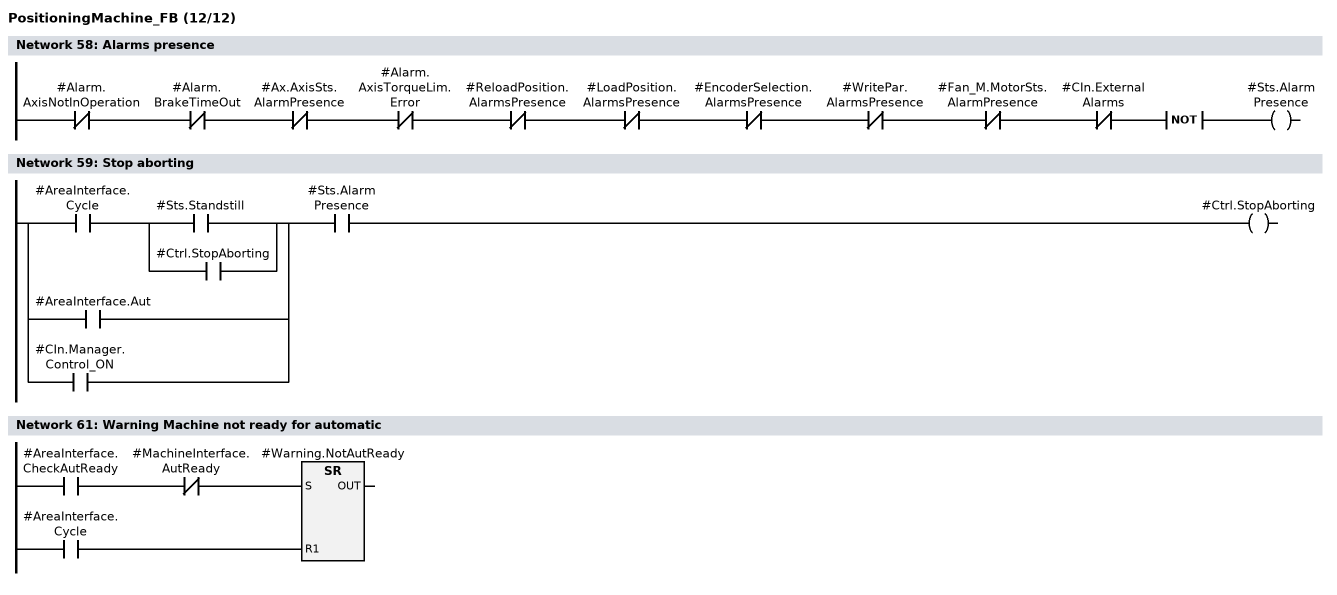
   RUNG wire#powerrail
      I_Contact( #Alarm.AxisNotInOperation )
      I_Contact( #Alarm.BrakeTimeOut )
      I_Contact( #Ax.AxisSts.AlarmPresence )
      I_Contact( #Alarm.AxisTorqueLim.Error )
      I_Contact( #ReloadPosition.AlarmsPresence )
      I_Contact( #LoadPosition.AlarmsPresence )
      I_Contact( #EncoderSelection.AlarmsPresence )
      I_Contact( #WritePar.AlarmsPresence )
      I_Contact( #Fan_M.MotorSts.AlarmPresence )
      I_Contact( #CIn.ExternalAlarms )
      Not()
      Coil( #Sts.AlarmPresence )
   END_RUNG
   // the same network as SCL:
   #Sts.AlarmPresence := NOT (NOT #Alarm.AxisNotInOperation AND NOT #Alarm.BrakeTimeOut AND NOT #Ax.AxisSts.AlarmPresence AND NOT #Alarm.AxisTorqueLim.Error AND NOT #ReloadPosition.AlarmsPresence AND NOT #LoadPosition.AlarmsPresence AND NOT #EncoderSelection.AlarmsPresence AND NOT #WritePar.AlarmsPresence AND NOT #Fan_M.MotorSts.AlarmPresence AND NOT #CIn.ExternalAlarms);
END_REGION

REGION Network 59: Stop aborting
   RUNG wire#powerrail
      Contact( #AreaInterface.Cycle )
      wire#w1
      Contact( #Sts.Standstill )
      wire#w2
      Contact( #Sts.AlarmPresence )
      Coil( #Ctrl.StopAborting )
   END_RUNG
   RUNG wire#w1
      Contact( #Ctrl.StopAborting )
   END_RUNG wire#w2
   RUNG wire#powerrail
      Contact( #AreaInterface.Aut )
   END_RUNG wire#w2
   RUNG wire#powerrail
      Contact( #CIn.Manager.Control_ON )
   END_RUNG wire#w2
   // the same network as SCL:
   #Ctrl.StopAborting := ((#AreaInterface.Cycle AND (#Sts.Standstill OR #Ctrl.StopAborting)) OR #AreaInterface.Aut OR #CIn.Manager.Control_ON) AND #Sts.AlarmPresence;
END_REGION

REGION Network 60 (SCL): Collect machine to zone interface
   #MachineInterface.AutReady := #AreaInterface.Aut AND NOT #Sts.AlarmPresence;
   #MachineInterface.Aborting := #Ctrl.StopAborting;
   #MachineInterface.MotionsStandStill := #TON_NoPendingCmd.Q AND #Sts.Standstill;
   #MachineInterface.AckStopInPhase := #Ctrl.StopInPhase AND #MachineInterface.MotionsStandStill;
   #MachineInterface.AckStopProgrammed := #Ctrl.StopProgrammed AND #MachineInterface.MotionsStandStill;
   #MachineInterface.AlarmsPresence := #Sts.AlarmPresence;
   #MachineInterface.WarningPresence := #Sts.WarningPresence;
END_REGION

REGION Network 61: Warning Machine not ready for automatic
   RUNG wire#powerrail
      Contact( #AreaInterface.CheckAutReady )
      I_Contact( #MachineInterface.AutReady )
      S_SR(operand := #Warning.NotAutReady, r1 := wire#w1)
   END_RUNG
   RUNG wire#powerrail
      Contact( #AreaInterface.Cycle )
   END_RUNG wire#w1
   // the same network as SCL:
   IF #AreaInterface.CheckAutReady AND NOT #MachineInterface.AutReady THEN
       #Warning.NotAutReady := TRUE;   // SR flip-flop
   END_IF;
   IF #AreaInterface.Cycle THEN #Warning.NotAutReady := FALSE; END_IF;
END_REGION

REGION Network 62 (SCL): ENO
   ENO := NOT #Sts.AlarmPresence;
END_REGION

REGION Network 63: >
END_REGION

REGION Network 64: >
END_REGION

REGION Network 65: >
END_REGION
END_FUNCTION_BLOCK
